LIN {X 0,Y 470.205,Z 358.727,A -85,B 0,C 180,E1 -7723.342,E2 -7723.342} C_VEL
LIN {X 0,Y 469.487,Z 370.693,A -85,B 0,C 180,E1 -7724.591,E2 -7724.591} C_VEL
LIN {X 0,Y 468.899,Z 381.216,A -85,B 0,C 180,E1 -7725.904,E2 -7725.904} C_VEL
LIN {X 0,Y 468.341,Z 390.427,A -85,B 0,C 180,E1 -7727.265,E2 -7727.265} C_VEL
LIN {X 0,Y 467.874,Z 398.79,A -85,B 0,C 180,E1 -7728.739,E2 -7728.739} C_VEL
LIN {X 0,Y 467.533,Z 405.048,A -85,B 0,C 180,E1 -7730.046,E2 -7730.046} C_VEL
LIN {X 0,Y 467.216,Z 411.873,A -85,B 0,C 180,E1 -7731.784,E2 -7731.784} C_VEL
LIN {X 0,Y 467.007,Z 416.636,A -85,B 0,C 180,E1 -7733.332,E2 -7733.332} C_VEL
LIN {X 0,Y 466.794,Z 420.207,A -85,B 0,C 180,E1 -7734.817,E2 -7734.817} C_VEL
LIN {X 0,Y 466.834,Z 423.167,A -85,B 0,C 180,E1 -7736.548,E2 -7736.548} C_VEL
LIN {X 0,Y 466.699,Z 424.922,A -85,B 0,C 180,E1 -7738.274,E2 -7738.274} C_VEL
LIN {X 0,Y 466.612,Z 425.477,A -85,B 0,C 180,E1 -7740,E2 -7740} C_VEL
LIN {X 0,Y 466.699,Z 424.809,A -85,B 0,C 180,E1 -7741.726,E2 -7741.726} C_VEL
LIN {X 0,Y 466.823,Z 422.958,A -85,B 0,C 180,E1 -7743.453,E2 -7743.453} C_VEL
LIN {X 0,Y 466.783,Z 419.896,A -85,B 0,C 180,E1 -7745.183,E2 -7745.183} C_VEL
LIN {X 0,Y 466.969,Z 416.065,A -85,B 0,C 180,E1 -7746.733,E2 -7746.733} C_VEL
LIN {X 0,Y 467.137,Z 411.402,A -85,B 0,C 180,E1 -7748.217,E2 -7748.217} C_VEL
LIN {X 0,Y 467.418,Z 404.499,A -85,B 0,C 180,E1 -7749.957,E2 -7749.957} C_VEL
LIN {X 0,Y 467.832,Z 397.038,A -85,B 0,C 180,E1 -7751.482,E2 -7751.482} C_VEL
LIN {X 0,Y 468.246,Z 388.039,A -85,B 0,C 180,E1 -7753.011,E2 -7753.011} C_VEL
LIN {X 0,Y 468.878,Z 377.174,A -85,B 0,C 180,E1 -7754.541,E2 -7754.541} C_VEL
LIN {X 0,Y 469.527,Z 365.967,A -85,B 0,C 180,E1 -7755.853,E2 -7755.853} C_VEL
LIN {X 0,Y 470.209,Z 354.013,A -85,B 0,C 180,E1 -7757.027,E2 -7757.027} C_VEL
LIN {X 0,Y 470.969,Z 340.123,A -85,B 0,C 180,E1 -7758.15,E2 -7758.15} C_VEL
LIN {X 0,Y 471.618,Z 326.912,A -85,B 0,C 180,E1 -7759.025,E2 -7759.025} C_VEL
LIN {X 0,Y 472.295,Z 312.467,A -85,B 0,C 180,E1 -7759.788,E2 -7759.788} C_VEL
LIN {X 0,Y 472.767,Z 297.672,A -85,B 0,C 180,E1 -7760.391,E2 -7760.391} C_VEL
LIN {X 0,Y 473.123,Z 282.745,A -85,B 0,C 180,E1 -7760.829,E2 -7760.829} C_VEL
LIN {X 0,Y 473.547,Z 255.622,A -85,B 0,C 180,E1 -7761.322,E2 -7761.322} C_VEL
LIN {X 0,Y 475.612,Z 134.89,A -85,B 0,C 180,E1 -7763.422,E2 -7763.422} C_VEL
LIN {X 0,Y 468.054,Z 114.952,A -85,B 0,C 180,E1 -7764.181,E2 -7764.181} C_VEL
LIN {X 0,Y 467.613,Z 112.864,A -85,B 0,C 180,E1 -7764.532,E2 -7764.532} C_VEL
LIN {X 0,Y 467.563,Z 112.87,A -85,B 0,C 180,E1 -7767.773,E2 -7767.773} C_VEL
LIN {X 0,Y 467.567,Z 112.867,A -85,B 0,C 180,E1 -7771.044,E2 -7771.044} C_VEL
LIN {X 0,Y 467.578,Z 112.864,A -85,B 0,C 180,E1 -7774.24,E2 -7774.24} C_VEL
LIN {X 0,Y 467.544,Z 112.871,A -85,B 0,C 180,E1 -7777.186,E2 -7777.186} C_VEL
LIN {X 0,Y 467.559,Z 112.865,A -85,B 0,C 180,E1 -7780.267,E2 -7780.267} C_VEL
LIN {X 0,Y 467.548,Z 112.866,A -85,B 0,C 180,E1 -7783.746,E2 -7783.746} C_VEL
LIN {X 0,Y 467.546,Z 112.852,A -85,B 0,C 180,E1 -7786.254,E2 -7786.254} C_VEL
LIN {X 0,Y 467.559,Z 112.867,A -85,B 0,C 180,E1 -7789.733,E2 -7789.733} C_VEL
LIN {X 0,Y 467.545,Z 112.869,A -85,B 0,C 180,E1 -7792.815,E2 -7792.815} C_VEL
LIN {X 0,Y 467.549,Z 112.855,A -85,B 0,C 180,E1 -7794.076,E2 -7794.076} C_VEL
LIN {X 0,Y 466.939,Z 112.935,A -85,B 0,C 180,E1 -7794.794,E2 -7794.794} C_VEL
LIN {X 0,Y 464.105,Z 113.293,A -85,B 0,C 180,E1 -7795.962,E2 -7795.962} C_VEL
LIN {X 0,Y 461.665,Z 113.603,A -85,B 0,C 180,E1 -7796.903,E2 -7796.903} C_VEL
LIN {X 0,Y 460.603,Z 113.733,A -85,B 0,C 180,E1 -7797.631,E2 -7797.631} C_VEL
LIN {X 0,Y 460.51,Z 113.743,A -85,B 0,C 180,E1 -7797.877,E2 -7797.877} C_VEL
LIN {X 0,Y 460.518,Z 113.738,A -85,B 0,C 180,E1 -7800.767,E2 -7800.767} C_VEL
LIN {X 0,Y 460.521,Z 113.743,A -85,B 0,C 180,E1 -7803.732,E2 -7803.732} C_VEL
LIN {X 0,Y 460.544,Z 113.737,A -85,B 0,C 180,E1 -7806.624,E2 -7806.624} C_VEL
LIN {X 0,Y 460.542,Z 113.737,A -85,B 0,C 180,E1 -7809.452,E2 -7809.452} C_VEL
LIN {X 0,Y 460.527,Z 113.745,A -85,B 0,C 180,E1 -7812.229,E2 -7812.229} C_VEL
LIN {X 0,Y 460.548,Z 113.743,A -85,B 0,C 180,E1 -7814.964,E2 -7814.964} C_VEL
LIN {X 0,Y 460.612,Z 113.736,A -85,B 0,C 180,E1 -7818.559,E2 -7818.559} C_VEL
LIN {X 0,Y 460.626,Z 113.732,A -85,B 0,C 180,E1 -7822.107,E2 -7822.107} C_VEL
LIN {X 0,Y 460.672,Z 113.729,A -85,B 0,C 180,E1 -7824.748,E2 -7824.748} C_VEL
LIN {X 0,Y 460.758,Z 113.718,A -85,B 0,C 180,E1 -7827.377,E2 -7827.377} C_VEL
LIN {X 0,Y 460.715,Z 113.854,A -85,B 0,C 180,E1 -7828.306,E2 -7828.306} C_VEL
LIN {X 0,Y 463.866,Z 127.486,A -85,B 0,C 180,E1 -7830.46,E2 -7830.46} C_VEL
LIN {X 0,Y 464.926,Z 132.74,A -85,B 0,C 180,E1 -7831.28,E2 -7831.28} C_VEL
LIN {X 0,Y 464.725,Z 142.504,A -85,B 0,C 180,E1 -7832.646,E2 -7832.646} C_VEL
LIN {X 0,Y 469.356,Z 164.409,A -85,B 0,C 180,E1 -7833.26,E2 -7833.26} C_VEL
LIN {X 0,Y 467.464,Z 308.671,A -85,B 0,C 180,E1 -7835.554,E2 -7835.554} C_VEL
LIN {X 0,Y 467.063,Z 323.846,A -85,B 0,C 180,E1 -7835.965,E2 -7835.965} C_VEL
LIN {X 0,Y 466.453,Z 338.982,A -85,B 0,C 180,E1 -7836.556,E2 -7836.556} C_VEL
LIN {X 0,Y 465.768,Z 352.68,A -85,B 0,C 180,E1 -7837.26,E2 -7837.26} C_VEL
LIN {X 0,Y 464.914,Z 366.405,A -85,B 0,C 180,E1 -7838.147,E2 -7838.147} C_VEL
LIN {X 0,Y 464.107,Z 378.997,A -85,B 0,C 180,E1 -7839.149,E2 -7839.149} C_VEL
LIN {X 0,Y 463.263,Z 390.836,A -85,B 0,C 180,E1 -7840.28,E2 -7840.28} C_VEL
LIN {X 0,Y 462.424,Z 402.5,A -85,B 0,C 180,E1 -7841.617,E2 -7841.617} C_VEL
LIN {X 0,Y 461.673,Z 412.766,A -85,B 0,C 180,E1 -7843.025,E2 -7843.025} C_VEL
LIN {X 0,Y 461.03,Z 422.16,A -85,B 0,C 180,E1 -7844.568,E2 -7844.568} C_VEL
LIN {X 0,Y 460.56,Z 429.373,A -85,B 0,C 180,E1 -7845.978,E2 -7845.978} C_VEL
LIN {X 0,Y 460.148,Z 436.979,A -85,B 0,C 180,E1 -7847.786,E2 -7847.786} C_VEL
LIN {X 0,Y 459.856,Z 443.115,A -85,B 0,C 180,E1 -7849.647,E2 -7849.647} C_VEL
LIN {X 0,Y 459.632,Z 447.79,A -85,B 0,C 180,E1 -7851.529,E2 -7851.529} C_VEL
LIN {X 0,Y 459.464,Z 451.071,A -85,B 0,C 180,E1 -7853.434,E2 -7853.434} C_VEL
LIN {X 0,Y 459.416,Z 452.973,A -85,B 0,C 180,E1 -7855.362,E2 -7855.362} C_VEL
LIN {X 0,Y 459.426,Z 453.492,A -85,B 0,C 180,E1 -7857.317,E2 -7857.317} C_VEL
LIN {X 0,Y 459.45,Z 452.559,A -85,B 0,C 180,E1 -7859.319,E2 -7859.319} C_VEL
LIN {X 0,Y 459.534,Z 450.116,A -85,B 0,C 180,E1 -7861.331,E2 -7861.331} C_VEL
LIN {X 0,Y 459.649,Z 447.476,A -85,B 0,C 180,E1 -7862.759,E2 -7862.759} C_VEL
LIN {X 0,Y 459.815,Z 443.254,A -85,B 0,C 180,E1 -7864.439,E2 -7864.439} C_VEL
LIN {X 0,Y 460.136,Z 437.453,A -85,B 0,C 180,E1 -7866.215,E2 -7866.215} C_VEL
LIN {X 0,Y 460.508,Z 430.544,A -85,B 0,C 180,E1 -7867.899,E2 -7867.899} C_VEL
LIN {X 0,Y 461.041,Z 422.167,A -85,B 0,C 180,E1 -7869.567,E2 -7869.567} C_VEL
LIN {X 0,Y 461.744,Z 412.393,A -85,B 0,C 180,E1 -7871.17,E2 -7871.17} C_VEL
LIN {X 0,Y 462.565,Z 401.147,A -85,B 0,C 180,E1 -7872.689,E2 -7872.689} C_VEL
LIN {X 0,Y 463.356,Z 389.986,A -85,B 0,C 180,E1 -7873.948,E2 -7873.948} C_VEL
LIN {X 0,Y 464.296,Z 377.438,A -85,B 0,C 180,E1 -7875.123,E2 -7875.123} C_VEL
LIN {X 0,Y 465.113,Z 364.512,A -85,B 0,C 180,E1 -7876.125,E2 -7876.125} C_VEL
LIN {X 0,Y 465.98,Z 350.355,A -85,B 0,C 180,E1 -7877.009,E2 -7877.009} C_VEL
LIN {X 0,Y 466.709,Z 336.007,A -85,B 0,C 180,E1 -7877.711,E2 -7877.711} C_VEL
LIN {X 0,Y 467.223,Z 320.852,A -85,B 0,C 180,E1 -7878.265,E2 -7878.265} C_VEL
LIN {X 0,Y 467.643,Z 306.467,A -85,B 0,C 180,E1 -7878.621,E2 -7878.621} C_VEL
LIN {X 0,Y 469.619,Z 160.081,A -85,B 0,C 180,E1 -7880.948,E2 -7880.948} C_VEL
LIN {X 0,Y 466.099,Z 140.754,A -85,B 0,C 180,E1 -7881.491,E2 -7881.491} C_VEL
LIN {X 0,Y 466.266,Z 135.208,A -85,B 0,C 180,E1 -7882.104,E2 -7882.104} C_VEL
LIN {X 0,Y 462.6,Z 121.002,A -85,B 0,C 180,E1 -7883.914,E2 -7883.914} C_VEL
LIN {X 0,Y 460.536,Z 113.744,A -85,B 0,C 180,E1 -7884.871,E2 -7884.871} C_VEL
LIN {X 0,Y 460.534,Z 113.747,A -85,B 0,C 180,E1 -7887.715,E2 -7887.715} C_VEL
LIN {X 0,Y 460.542,Z 113.739,A -85,B 0,C 180,E1 -7890.769,E2 -7890.769} C_VEL
LIN {X 0,Y 460.566,Z 113.742,A -85,B 0,C 180,E1 -7893.735,E2 -7893.735} C_VEL
LIN {X 0,Y 460.57,Z 113.75,A -85,B 0,C 180,E1 -7895.369,E2 -7895.369} C_VEL
LIN {X 0,Y 460.779,Z 114.732,A -85,B 0,C 180,E1 -7895.514,E2 -7895.514} C_VEL
LIN {X 0,Y 469.062,Z 135.535,A -85,B 0,C 180,E1 -7896.336,E2 -7896.336} C_VEL
LIN {X 0,Y 466.423,Z 282.486,A -85,B 0,C 180,E1 -7898.977,E2 -7898.977} C_VEL
LIN {X 0,Y 466.028,Z 297.981,A -85,B 0,C 180,E1 -7899.434,E2 -7899.434} C_VEL
LIN {X 0,Y 465.501,Z 312.425,A -85,B 0,C 180,E1 -7900.026,E2 -7900.026} C_VEL
LIN {X 0,Y 464.802,Z 326.942,A -85,B 0,C 180,E1 -7900.8,E2 -7900.8} C_VEL
LIN {X 0,Y 464.134,Z 340.27,A -85,B 0,C 180,E1 -7901.687,E2 -7901.687} C_VEL
LIN {X 0,Y 463.457,Z 352.85,A -85,B 0,C 180,E1 -7902.706,E2 -7902.706} C_VEL
LIN {X 0,Y 462.676,Z 365.193,A -85,B 0,C 180,E1 -7903.906,E2 -7903.906} C_VEL
LIN {X 0,Y 462.018,Z 376.615,A -85,B 0,C 180,E1 -7905.238,E2 -7905.238} C_VEL
LIN {X 0,Y 461.33,Z 387.666,A -85,B 0,C 180,E1 -7906.79,E2 -7906.79} C_VEL
LIN {X 0,Y 460.873,Z 396.82,A -85,B 0,C 180,E1 -7908.343,E2 -7908.343} C_VEL
LIN {X 0,Y 460.423,Z 404.413,A -85,B 0,C 180,E1 -7909.89,E2 -7909.89} C_VEL
LIN {X 0,Y 460.104,Z 411.459,A -85,B 0,C 180,E1 -7911.656,E2 -7911.656} C_VEL
LIN {X 0,Y 459.861,Z 416.937,A -85,B 0,C 180,E1 -7913.408,E2 -7913.408} C_VEL
LIN {X 0,Y 459.736,Z 420.149,A -85,B 0,C 180,E1 -7914.737,E2 -7914.737} C_VEL
LIN {X 0,Y 459.76,Z 423.312,A -85,B 0,C 180,E1 -7916.494,E2 -7916.494} C_VEL
LIN {X 0,Y 459.638,Z 425.267,A -85,B 0,C 180,E1 -7918.247,E2 -7918.247} C_VEL
LIN {X 0,Y 459.545,Z 426.009,A -85,B 0,C 180,E1 -7920,E2 -7920} C_VEL
LIN {X 0,Y 459.639,Z 425.528,A -85,B 0,C 180,E1 -7921.752,E2 -7921.752} C_VEL
LIN {X 0,Y 459.777,Z 423.863,A -85,B 0,C 180,E1 -7923.505,E2 -7923.505} C_VEL
LIN {X 0,Y 459.749,Z 420.99,A -85,B 0,C 180,E1 -7925.262,E2 -7925.262} C_VEL
LIN {X 0,Y 460.008,Z 417.57,A -85,B 0,C 180,E1 -7926.749,E2 -7926.749} C_VEL
LIN {X 0,Y 460.19,Z 412.788,A -85,B 0,C 180,E1 -7928.342,E2 -7928.342} C_VEL
LIN {X 0,Y 460.528,Z 406.086,A -85,B 0,C 180,E1 -7930.107,E2 -7930.107} C_VEL
LIN {X 0,Y 460.97,Z 398.787,A -85,B 0,C 180,E1 -7931.654,E2 -7931.654} C_VEL
LIN {X 0,Y 461.482,Z 389.975,A -85,B 0,C 180,E1 -7933.205,E2 -7933.205} C_VEL
LIN {X 0,Y 462.121,Z 380.966,A -85,B 0,C 180,E1 -7934.533,E2 -7934.533} C_VEL
LIN {X 0,Y 462.797,Z 370.287,A -85,B 0,C 180,E1 -7935.863,E2 -7935.863} C_VEL
LIN {X 0,Y 463.608,Z 357.669,A -85,B 0,C 180,E1 -7937.173,E2 -7937.173} C_VEL
LIN {X 0,Y 464.377,Z 344.479,A -85,B 0,C 180,E1 -7938.302,E2 -7938.302} C_VEL
LIN {X 0,Y 465.093,Z 331.89,A -85,B 0,C 180,E1 -7939.187,E2 -7939.187} C_VEL
LIN {X 0,Y 465.707,Z 318.4,A -85,B 0,C 180,E1 -7939.964,E2 -7939.964} C_VEL
LIN {X 0,Y 466.334,Z 302.907,A -85,B 0,C 180,E1 -7940.654,E2 -7940.654} C_VEL
LIN {X 0,Y 466.798,Z 287.065,A -85,B 0,C 180,E1 -7941.165,E2 -7941.165} C_VEL
LIN {X 0,Y 467.313,Z 262.068,A -85,B 0,C 180,E1 -7941.678,E2 -7941.678} C_VEL
LIN {X 0,Y 469.548,Z 178.96,A -85,B 0,C 180,E1 -7943.33,E2 -7943.33} C_VEL
LIN {X 0,Y 470.871,Z 139.064,A -85,B 0,C 180,E1 -7944.172,E2 -7944.172} C_VEL
LIN {X 0,Y 465.458,Z 127.422,A -85,B 0,C 180,E1 -7944.861,E2 -7944.861} C_VEL
LIN {X 0,Y 462.823,Z 122.223,A -85,B 0,C 180,E1 -7945.225,E2 -7945.225} C_VEL
LIN {X 0,Y 460.525,Z 113.749,A -85,B 0,C 180,E1 -7947.45,E2 -7947.45} C_VEL
LIN {X 0,Y 460.504,Z 113.75,A -85,B 0,C 180,E1 -7950.24,E2 -7950.24} C_VEL
LIN {X 0,Y 460.516,Z 113.748,A -85,B 0,C 180,E1 -7953.326,E2 -7953.326} C_VEL
LIN {X 0,Y 460.472,Z 113.752,A -85,B 0,C 180,E1 -7956.53,E2 -7956.53} C_VEL
LIN {X 0,Y 460.513,Z 113.748,A -85,B 0,C 180,E1 -7959.864,E2 -7959.864} C_VEL
LIN {X 0,Y 460.461,Z 113.754,A -85,B 0,C 180,E1 -7962.893,E2 -7962.893} C_VEL
LIN {X 0,Y 460.502,Z 113.748,A -85,B 0,C 180,E1 -7965.831,E2 -7965.831} C_VEL
LIN {X 0,Y 460.513,Z 113.749,A -85,B 0,C 180,E1 -7968.987,E2 -7968.987} C_VEL
LIN {X 0,Y 460.497,Z 113.751,A -85,B 0,C 180,E1 -7972.376,E2 -7972.376} C_VEL
LIN {X 0,Y 460.534,Z 113.747,A -85,B 0,C 180,E1 -7975.623,E2 -7975.623} C_VEL
LIN {X 0,Y 460.531,Z 113.873,A -85,B 0,C 180,E1 -7976.854,E2 -7976.854} C_VEL
LIN {X 0,Y 463.777,Z 124.861,A -85,B 0,C 180,E1 -7979.198,E2 -7979.198} C_VEL
LIN {X 0,Y 466.239,Z 135.335,A -85,B 0,C 180,E1 -7981.16,E2 -7981.16} C_VEL
LIN {X 0,Y 466.332,Z 138.39,A -85,B 0,C 180,E1 -7981.658,E2 -7981.658} C_VEL
LIN {X 0,Y 464.916,Z 155.637,A -85,B 0,C 180,E1 -7984.24,E2 -7984.24} C_VEL
LIN {X 0,Y 464.589,Z 160.323,A -85,B 0,C 180,E1 -7984.925,E2 -7984.925} C_VEL
LIN {X 0,Y 468.206,Z 179.445,A -85,B 0,C 180,E1 -7985.649,E2 -7985.649} C_VEL
LIN {X 0,Y 469.863,Z 191.952,A -85,B 0,C 180,E1 -7986.049,E2 -7986.049} C_VEL
LIN {X 0,Y 467.42,Z 282.385,A -85,B 0,C 180,E1 -7987.862,E2 -7987.862} C_VEL
LIN {X 0,Y 466.4,Z 330.968,A -85,B 0,C 180,E1 -7988.799,E2 -7988.799} C_VEL
LIN {X 0,Y 465.612,Z 350.742,A -85,B 0,C 180,E1 -7989.39,E2 -7989.39} C_VEL
LIN {X 0,Y 465.03,Z 366.077,A -85,B 0,C 180,E1 -7990.005,E2 -7990.005} C_VEL
LIN {X 0,Y 464.275,Z 380.562,A -85,B 0,C 180,E1 -7990.777,E2 -7990.777} C_VEL
LIN {X 0,Y 463.575,Z 393.745,A -85,B 0,C 180,E1 -7991.665,E2 -7991.665} C_VEL
LIN {X 0,Y 462.845,Z 405.936,A -85,B 0,C 180,E1 -7992.663,E2 -7992.663} C_VEL
LIN {X 0,Y 461.989,Z 418.546,A -85,B 0,C 180,E1 -7993.912,E2 -7993.912} C_VEL
LIN {X 0,Y 461.396,Z 429.488,A -85,B 0,C 180,E1 -7995.218,E2 -7995.218} C_VEL
LIN {X 0,Y 460.854,Z 438.906,A -85,B 0,C 180,E1 -7996.552,E2 -7996.552} C_VEL
LIN {X 0,Y 460.304,Z 448.353,A -85,B 0,C 180,E1 -7998.146,E2 -7998.146} C_VEL
LIN {X 0,Y 460.037,Z 455.754,A -85,B 0,C 180,E1 -7999.659,E2 -7999.659} C_VEL
LIN {X 0,Y 459.802,Z 462.035,A -85,B 0,C 180,E1 -8001.208,E2 -8001.208} C_VEL
LIN {X 0,Y 459.725,Z 467.769,A -85,B 0,C 180,E1 -8002.975,E2 -8002.975} C_VEL
LIN {X 0,Y 459.626,Z 472.092,A -85,B 0,C 180,E1 -8004.736,E2 -8004.736} C_VEL
LIN {X 0,Y 459.595,Z 475.12,A -85,B 0,C 180,E1 -8006.493,E2 -8006.493} C_VEL
LIN {X 0,Y 459.598,Z 476.93,A -85,B 0,C 180,E1 -8008.247,E2 -8008.247} C_VEL
LIN {X 0,Y 459.536,Z 477.546,A -85,B 0,C 180,E1 -8010,E2 -8010} C_VEL
LIN {X 0,Y 459.597,Z 476.948,A -85,B 0,C 180,E1 -8011.753,E2 -8011.753} C_VEL
LIN {X 0,Y 459.608,Z 475.152,A -85,B 0,C 180,E1 -8013.507,E2 -8013.507} C_VEL
LIN {X 0,Y 459.63,Z 472.125,A -85,B 0,C 180,E1 -8015.264,E2 -8015.264} C_VEL
LIN {X 0,Y 459.727,Z 467.802,A -85,B 0,C 180,E1 -8017.025,E2 -8017.025} C_VEL
LIN {X 0,Y 459.802,Z 462.075,A -85,B 0,C 180,E1 -8018.792,E2 -8018.792} C_VEL
LIN {X 0,Y 460.128,Z 454.78,A -85,B 0,C 180,E1 -8020.561,E2 -8020.561} C_VEL
LIN {X 0,Y 460.382,Z 446.748,A -85,B 0,C 180,E1 -8022.146,E2 -8022.146} C_VEL
LIN {X 0,Y 460.882,Z 437.413,A -85,B 0,C 180,E1 -8023.672,E2 -8023.672} C_VEL
LIN {X 0,Y 461.45,Z 427.686,A -85,B 0,C 180,E1 -8025.006,E2 -8025.006} C_VEL
LIN {X 0,Y 462.107,Z 416.662,A -85,B 0,C 180,E1 -8026.278,E2 -8026.278} C_VEL
LIN {X 0,Y 462.801,Z 404.49,A -85,B 0,C 180,E1 -8027.453,E2 -8027.453} C_VEL
LIN {X 0,Y 463.626,Z 391.995,A -85,B 0,C 180,E1 -8028.448,E2 -8028.448} C_VEL
LIN {X 0,Y 464.369,Z 378.323,A -85,B 0,C 180,E1 -8029.334,E2 -8029.334} C_VEL
LIN {X 0,Y 465.059,Z 364.285,A -85,B 0,C 180,E1 -8030.051,E2 -8030.051} C_VEL
LIN {X 0,Y 465.774,Z 346.56,A -85,B 0,C 180,E1 -8030.748,E2 -8030.748} C_VEL
LIN {X 0,Y 466.243,Z 330.73,A -85,B 0,C 180,E1 -8031.184,E2 -8031.184} C_VEL
LIN {X 0,Y 468.656,Z 202.97,A -85,B 0,C 180,E1 -8033.474,E2 -8033.474} C_VEL
LIN {X 0,Y 468.982,Z 186.436,A -85,B 0,C 180,E1 -8033.833,E2 -8033.833} C_VEL
LIN {X 0,Y 465.653,Z 160.353,A -85,B 0,C 180,E1 -8034.701,E2 -8034.701} C_VEL
LIN {X 0,Y 466.909,Z 137.343,A -85,B 0,C 180,E1 -8037.197,E2 -8037.197} C_VEL
LIN {X 0,Y 462.077,Z 119.489,A -85,B 0,C 180,E1 -8039.494,E2 -8039.494} C_VEL
LIN {X 0,Y 460.535,Z 113.746,A -85,B 0,C 180,E1 -8040.27,E2 -8040.27} C_VEL
LIN {X 0,Y 460.515,Z 113.748,A -85,B 0,C 180,E1 -8043.326,E2 -8043.326} C_VEL
LIN {X 0,Y 460.471,Z 113.754,A -85,B 0,C 180,E1 -8046.53,E2 -8046.53} C_VEL
LIN {X 0,Y 460.512,Z 113.746,A -85,B 0,C 180,E1 -8049.865,E2 -8049.865} C_VEL
LIN {X 0,Y 460.461,Z 113.755,A -85,B 0,C 180,E1 -8052.894,E2 -8052.894} C_VEL
LIN {X 0,Y 460.502,Z 113.743,A -85,B 0,C 180,E1 -8055.832,E2 -8055.832} C_VEL
LIN {X 0,Y 460.514,Z 113.745,A -85,B 0,C 180,E1 -8058.987,E2 -8058.987} C_VEL
LIN {X 0,Y 460.497,Z 113.75,A -85,B 0,C 180,E1 -8062.377,E2 -8062.377} C_VEL
LIN {X 0,Y 460.535,Z 113.743,A -85,B 0,C 180,E1 -8065.623,E2 -8065.623} C_VEL
LIN {X 0,Y 460.537,Z 113.746,A -85,B 0,C 180,E1 -8068.745,E2 -8068.745} C_VEL
LIN {X 0,Y 460.531,Z 113.748,A -85,B 0,C 180,E1 -8072.266,E2 -8072.266} C_VEL
LIN {X 0,Y 460.539,Z 113.891,A -85,B 0,C 180,E1 -8073.84,E2 -8073.84} C_VEL
LIN {X 0,Y 462.385,Z 119.757,A -85,B 0,C 180,E1 -8074.851,E2 -8074.851} C_VEL
LIN {X 0,Y 468.701,Z 132.928,A -85,B 0,C 180,E1 -8075.669,E2 -8075.669} C_VEL
LIN {X 0,Y 470.74,Z 137.876,A -85,B 0,C 180,E1 -8075.936,E2 -8075.936} C_VEL
LIN {X 0,Y 468.083,Z 226.35,A -85,B 0,C 180,E1 -8077.75,E2 -8077.75} C_VEL
LIN {X 0,Y 466.781,Z 285.261,A -85,B 0,C 180,E1 -8078.901,E2 -8078.901} C_VEL
LIN {X 0,Y 466.28,Z 301.493,A -85,B 0,C 180,E1 -8079.4,E2 -8079.4} C_VEL
LIN {X 0,Y 465.757,Z 316.216,A -85,B 0,C 180,E1 -8080.038,E2 -8080.038} C_VEL
LIN {X 0,Y 465.121,Z 330.113,A -85,B 0,C 180,E1 -8080.814,E2 -8080.814} C_VEL
LIN {X 0,Y 464.351,Z 344.421,A -85,B 0,C 180,E1 -8081.811,E2 -8081.811} C_VEL
LIN {X 0,Y 463.594,Z 356.511,A -85,B 0,C 180,E1 -8082.832,E2 -8082.832} C_VEL
LIN {X 0,Y 462.747,Z 369.234,A -85,B 0,C 180,E1 -8084.135,E2 -8084.135} C_VEL
LIN {X 0,Y 462.156,Z 380.059,A -85,B 0,C 180,E1 -8085.469,E2 -8085.469} C_VEL
LIN {X 0,Y 461.53,Z 389.205,A -85,B 0,C 180,E1 -8086.797,E2 -8086.797} C_VEL
LIN {X 0,Y 460.987,Z 398.127,A -85,B 0,C 180,E1 -8088.346,E2 -8088.346} C_VEL
LIN {X 0,Y 460.539,Z 405.491,A -85,B 0,C 180,E1 -8089.893,E2 -8089.893} C_VEL
LIN {X 0,Y 460.18,Z 412.311,A -85,B 0,C 180,E1 -8091.658,E2 -8091.658} C_VEL
LIN {X 0,Y 459.964,Z 417.265,A -85,B 0,C 180,E1 -8093.298,E2 -8093.298} C_VEL
LIN {X 0,Y 459.738,Z 420.64,A -85,B 0,C 180,E1 -8094.738,E2 -8094.738} C_VEL
LIN {X 0,Y 459.765,Z 423.589,A -85,B 0,C 180,E1 -8096.495,E2 -8096.495} C_VEL
LIN {X 0,Y 459.639,Z 425.328,A -85,B 0,C 180,E1 -8098.248,E2 -8098.248} C_VEL
LIN {X 0,Y 459.543,Z 425.869,A -85,B 0,C 180,E1 -8100,E2 -8100} C_VEL
LIN {X 0,Y 459.637,Z 425.178,A -85,B 0,C 180,E1 -8101.753,E2 -8101.753} C_VEL
LIN {X 0,Y 459.752,Z 423.296,A -85,B 0,C 180,E1 -8103.506,E2 -8103.506} C_VEL
LIN {X 0,Y 459.729,Z 420.196,A -85,B 0,C 180,E1 -8105.263,E2 -8105.263} C_VEL
LIN {X 0,Y 459.921,Z 415.793,A -85,B 0,C 180,E1 -8107.022,E2 -8107.022} C_VEL
LIN {X 0,Y 460.143,Z 409.989,A -85,B 0,C 180,E1 -8108.786,E2 -8108.786} C_VEL
LIN {X 0,Y 460.465,Z 402.615,A -85,B 0,C 180,E1 -8110.554,E2 -8110.554} C_VEL
LIN {X 0,Y 460.921,Z 394.673,A -85,B 0,C 180,E1 -8112.103,E2 -8112.103} C_VEL
LIN {X 0,Y 461.438,Z 385.101,A -85,B 0,C 180,E1 -8113.655,E2 -8113.655} C_VEL
LIN {X 0,Y 462.059,Z 375.307,A -85,B 0,C 180,E1 -8114.986,E2 -8114.986} C_VEL
LIN {X 0,Y 462.777,Z 363.644,A -85,B 0,C 180,E1 -8116.317,E2 -8116.317} C_VEL
LIN {X 0,Y 463.519,Z 350.687,A -85,B 0,C 180,E1 -8117.548,E2 -8117.548} C_VEL
LIN {X 0,Y 464.205,Z 338.078,A -85,B 0,C 180,E1 -8118.539,E2 -8118.539} C_VEL
LIN {X 0,Y 464.921,Z 324.287,A -85,B 0,C 180,E1 -8119.425,E2 -8119.425} C_VEL
LIN {X 0,Y 465.578,Z 309.007,A -85,B 0,C 180,E1 -8120.201,E2 -8120.201} C_VEL
LIN {X 0,Y 466.048,Z 293.672,A -85,B 0,C 180,E1 -8120.787,E2 -8120.787} C_VEL
LIN {X 0,Y 466.444,Z 277.954,A -85,B 0,C 180,E1 -8121.2,E2 -8121.2} C_VEL
LIN {X 0,Y 469.059,Z 137.414,A -85,B 0,C 180,E1 -8123.698,E2 -8123.698} C_VEL
LIN {X 0,Y 468.467,Z 134.85,A -85,B 0,C 180,E1 -8123.776,E2 -8123.776} C_VEL
LIN {X 0,Y 460.88,Z 115.188,A -85,B 0,C 180,E1 -8124.551,E2 -8124.551} C_VEL
LIN {X 0,Y 460.553,Z 113.743,A -85,B 0,C 180,E1 -8124.813,E2 -8124.813} C_VEL
LIN {X 0,Y 460.516,Z 113.746,A -85,B 0,C 180,E1 -8128.236,E2 -8128.236} C_VEL
LIN {X 0,Y 460.522,Z 113.746,A -85,B 0,C 180,E1 -8131.283,E2 -8131.283} C_VEL
LIN {X 0,Y 460.523,Z 113.742,A -85,B 0,C 180,E1 -8134.504,E2 -8134.504} C_VEL
LIN {X 0,Y 460.5,Z 113.75,A -85,B 0,C 180,E1 -8137.624,E2 -8137.624} C_VEL
LIN {X 0,Y 460.517,Z 113.745,A -85,B 0,C 180,E1 -8141.013,E2 -8141.013} C_VEL
LIN {X 0,Y 460.514,Z 113.74,A -85,B 0,C 180,E1 -8144.59,E2 -8144.59} C_VEL
LIN {X 0,Y 460.477,Z 113.743,A -85,B 0,C 180,E1 -8147.813,E2 -8147.813} C_VEL
LIN {X 0,Y 460.515,Z 113.743,A -85,B 0,C 180,E1 -8150.136,E2 -8150.136} C_VEL
LIN {X 0,Y 460.475,Z 113.739,A -85,B 0,C 180,E1 -8153.47,E2 -8153.47} C_VEL
LIN {X 0,Y 460.519,Z 113.743,A -85,B 0,C 180,E1 -8156.674,E2 -8156.674} C_VEL
LIN {X 0,Y 460.51,Z 113.743,A -85,B 0,C 180,E1 -8157.877,E2 -8157.877} C_VEL
LIN {X 0,Y 459.825,Z 113.832,A -85,B 0,C 180,E1 -8158.608,E2 -8158.608} C_VEL
LIN {X 0,Y 456.959,Z 114.185,A -85,B 0,C 180,E1 -8159.793,E2 -8159.793} C_VEL
LIN {X 0,Y 454.555,Z 114.483,A -85,B 0,C 180,E1 -8160.75,E2 -8160.75} C_VEL
LIN {X 0,Y 453.538,Z 114.611,A -85,B 0,C 180,E1 -8161.489,E2 -8161.489} C_VEL
LIN {X 0,Y 453.462,Z 114.619,A -85,B 0,C 180,E1 -8161.739,E2 -8161.739} C_VEL
LIN {X 0,Y 453.496,Z 114.62,A -85,B 0,C 180,E1 -8164.283,E2 -8164.283} C_VEL
LIN {X 0,Y 453.476,Z 114.622,A -85,B 0,C 180,E1 -8167.204,E2 -8167.204} C_VEL
LIN {X 0,Y 453.498,Z 114.615,A -85,B 0,C 180,E1 -8170.066,E2 -8170.066} C_VEL
LIN {X 0,Y 453.475,Z 114.621,A -85,B 0,C 180,E1 -8172.875,E2 -8172.875} C_VEL
LIN {X 0,Y 453.498,Z 114.619,A -85,B 0,C 180,E1 -8175.643,E2 -8175.643} C_VEL
LIN {X 0,Y 453.561,Z 114.616,A -85,B 0,C 180,E1 -8178.379,E2 -8178.379} C_VEL
LIN {X 0,Y 453.564,Z 114.61,A -85,B 0,C 180,E1 -8181.086,E2 -8181.086} C_VEL
LIN {X 0,Y 453.631,Z 114.604,A -85,B 0,C 180,E1 -8183.774,E2 -8183.774} C_VEL
LIN {X 0,Y 453.689,Z 114.602,A -85,B 0,C 180,E1 -8187.781,E2 -8187.781} C_VEL
LIN {X 0,Y 453.729,Z 114.857,A -85,B 0,C 180,E1 -8188.003,E2 -8188.003} C_VEL
LIN {X 0,Y 456.825,Z 128.141,A -85,B 0,C 180,E1 -8190.133,E2 -8190.133} C_VEL
LIN {X 0,Y 458.173,Z 135.454,A -85,B 0,C 180,E1 -8191.273,E2 -8191.273} C_VEL
LIN {X 0,Y 457.986,Z 142.634,A -85,B 0,C 180,E1 -8192.275,E2 -8192.275} C_VEL
LIN {X 0,Y 462.797,Z 164.858,A -85,B 0,C 180,E1 -8192.918,E2 -8192.918} C_VEL
LIN {X 0,Y 460.877,Z 307.956,A -85,B 0,C 180,E1 -8195.222,E2 -8195.222} C_VEL
LIN {X 0,Y 460.434,Z 323.473,A -85,B 0,C 180,E1 -8195.639,E2 -8195.639} C_VEL
LIN {X 0,Y 459.818,Z 338.413,A -85,B 0,C 180,E1 -8196.222,E2 -8196.222} C_VEL
LIN {X 0,Y 459.049,Z 352.935,A -85,B 0,C 180,E1 -8196.975,E2 -8196.975} C_VEL
LIN {X 0,Y 458.223,Z 365.957,A -85,B 0,C 180,E1 -8197.823,E2 -8197.823} C_VEL
LIN {X 0,Y 457.307,Z 378.703,A -85,B 0,C 180,E1 -8198.84,E2 -8198.84} C_VEL
LIN {X 0,Y 456.431,Z 391.056,A -85,B 0,C 180,E1 -8200.037,E2 -8200.037} C_VEL
LIN {X 0,Y 455.558,Z 402.338,A -85,B 0,C 180,E1 -8201.344,E2 -8201.344} C_VEL
LIN {X 0,Y 454.76,Z 412.8,A -85,B 0,C 180,E1 -8202.794,E2 -8202.794} C_VEL
LIN {X 0,Y 454.073,Z 422.108,A -85,B 0,C 180,E1 -8204.338,E2 -8204.338} C_VEL
LIN {X 0,Y 453.48,Z 430.751,A -85,B 0,C 180,E1 -8206.08,E2 -8206.08} C_VEL
LIN {X 0,Y 453.122,Z 437,A -85,B 0,C 180,E1 -8207.605,E2 -8207.605} C_VEL
LIN {X 0,Y 452.787,Z 443.183,A -85,B 0,C 180,E1 -8209.494,E2 -8209.494} C_VEL
LIN {X 0,Y 452.586,Z 447.671,A -85,B 0,C 180,E1 -8211.296,E2 -8211.296} C_VEL
LIN {X 0,Y 452.355,Z 451.47,A -85,B 0,C 180,E1 -8213.557,E2 -8213.557} C_VEL
LIN {X 0,Y 452.297,Z 452.77,A -85,B 0,C 180,E1 -8214.805,E2 -8214.805} C_VEL
LIN {X 0,Y 452.292,Z 453.676,A -85,B 0,C 180,E1 -8216.784,E2 -8216.784} C_VEL
LIN {X 0,Y 452.318,Z 453.164,A -85,B 0,C 180,E1 -8218.795,E2 -8218.795} C_VEL
LIN {X 0,Y 452.381,Z 452.354,A -85,B 0,C 180,E1 -8219.811,E2 -8219.811} C_VEL
LIN {X 0,Y 452.456,Z 450.439,A -85,B 0,C 180,E1 -8221.315,E2 -8221.315} C_VEL
LIN {X 0,Y 452.574,Z 447.3,A -85,B 0,C 180,E1 -8223.011,E2 -8223.011} C_VEL
LIN {X 0,Y 452.782,Z 443.197,A -85,B 0,C 180,E1 -8224.648,E2 -8224.648} C_VEL
LIN {X 0,Y 453.061,Z 438.095,A -85,B 0,C 180,E1 -8226.231,E2 -8226.231} C_VEL
LIN {X 0,Y 453.491,Z 431.052,A -85,B 0,C 180,E1 -8227.997,E2 -8227.997} C_VEL
LIN {X 0,Y 454.028,Z 422.797,A -85,B 0,C 180,E1 -8229.681,E2 -8229.681} C_VEL
LIN {X 0,Y 454.714,Z 414.167,A -85,B 0,C 180,E1 -8231.141,E2 -8231.141} C_VEL
LIN {X 0,Y 455.51,Z 404.027,A -85,B 0,C 180,E1 -8232.584,E2 -8232.584} C_VEL
LIN {X 0,Y 456.309,Z 393.256,A -85,B 0,C 180,E1 -8233.875,E2 -8233.875} C_VEL
LIN {X 0,Y 457.322,Z 380.551,A -85,B 0,C 180,E1 -8235.14,E2 -8235.14} C_VEL
LIN {X 0,Y 458.196,Z 368.559,A -85,B 0,C 180,E1 -8236.129,E2 -8236.129} C_VEL
LIN {X 0,Y 459.09,Z 354.506,A -85,B 0,C 180,E1 -8237.079,E2 -8237.079} C_VEL
LIN {X 0,Y 459.877,Z 339.71,A -85,B 0,C 180,E1 -8237.867,E2 -8237.867} C_VEL
LIN {X 0,Y 460.535,Z 324.752,A -85,B 0,C 180,E1 -8238.464,E2 -8238.464} C_VEL
LIN {X 0,Y 460.986,Z 310.334,A -85,B 0,C 180,E1 -8238.866,E2 -8238.866} C_VEL
LIN {X 0,Y 461.501,Z 274.997,A -85,B 0,C 180,E1 -8239.464,E2 -8239.464} C_VEL
LIN {X 0,Y 463.152,Z 160.953,A -85,B 0,C 180,E1 -8241.297,E2 -8241.297} C_VEL
LIN {X 0,Y 459.475,Z 141.081,A -85,B 0,C 180,E1 -8241.861,E2 -8241.861} C_VEL
LIN {X 0,Y 459.608,Z 137.252,A -85,B 0,C 180,E1 -8242.291,E2 -8242.291} C_VEL
LIN {X 0,Y 455.424,Z 121.16,A -85,B 0,C 180,E1 -8244.37,E2 -8244.37} C_VEL
LIN {X 0,Y 453.515,Z 114.618,A -85,B 0,C 180,E1 -8245.262,E2 -8245.262} C_VEL
LIN {X 0,Y 453.468,Z 114.623,A -85,B 0,C 180,E1 -8248.475,E2 -8248.475} C_VEL
LIN {X 0,Y 453.535,Z 114.617,A -85,B 0,C 180,E1 -8252.04,E2 -8252.04} C_VEL
LIN {X 0,Y 453.568,Z 114.799,A -85,B 0,C 180,E1 -8255.116,E2 -8255.116} C_VEL
LIN {X 0,Y 462.415,Z 137.148,A -85,B 0,C 180,E1 -8256.037,E2 -8256.037} C_VEL
LIN {X 0,Y 459.988,Z 263.498,A -85,B 0,C 180,E1 -8258.341,E2 -8258.341} C_VEL
LIN {X 0,Y 459.621,Z 285.247,A -85,B 0,C 180,E1 -8258.78,E2 -8258.78} C_VEL
LIN {X 0,Y 459.198,Z 300.216,A -85,B 0,C 180,E1 -8259.253,E2 -8259.253} C_VEL
LIN {X 0,Y 458.594,Z 314.869,A -85,B 0,C 180,E1 -8259.888,E2 -8259.888} C_VEL
LIN {X 0,Y 457.85,Z 329.826,A -85,B 0,C 180,E1 -8260.729,E2 -8260.729} C_VEL
LIN {X 0,Y 457.037,Z 344.121,A -85,B 0,C 180,E1 -8261.741,E2 -8261.741} C_VEL
LIN {X 0,Y 456.333,Z 357.148,A -85,B 0,C 180,E1 -8262.873,E2 -8262.873} C_VEL
LIN {X 0,Y 455.555,Z 368.983,A -85,B 0,C 180,E1 -8264.107,E2 -8264.107} C_VEL
LIN {X 0,Y 454.889,Z 379.857,A -85,B 0,C 180,E1 -8265.459,E2 -8265.459} C_VEL
LIN {X 0,Y 454.221,Z 390.073,A -85,B 0,C 180,E1 -8266.975,E2 -8266.975} C_VEL
LIN {X 0,Y 453.757,Z 399.192,A -85,B 0,C 180,E1 -8268.61,E2 -8268.61} C_VEL
LIN {X 0,Y 453.298,Z 406.451,A -85,B 0,C 180,E1 -8270.18,E2 -8270.18} C_VEL
LIN {X 0,Y 452.995,Z 413.159,A -85,B 0,C 180,E1 -8271.973,E2 -8271.973} C_VEL
LIN {X 0,Y 452.811,Z 418.365,A -85,B 0,C 180,E1 -8273.762,E2 -8273.762} C_VEL
LIN {X 0,Y 452.631,Z 422.217,A -85,B 0,C 180,E1 -8275.547,E2 -8275.547} C_VEL
LIN {X 0,Y 452.632,Z 424.804,A -85,B 0,C 180,E1 -8277.33,E2 -8277.33} C_VEL
LIN {X 0,Y 452.498,Z 426.187,A -85,B 0,C 180,E1 -8279.11,E2 -8279.11} C_VEL
LIN {X 0,Y 452.499,Z 426.333,A -85,B 0,C 180,E1 -8280.89,E2 -8280.89} C_VEL
LIN {X 0,Y 452.673,Z 425.279,A -85,B 0,C 180,E1 -8282.669,E2 -8282.669} C_VEL
LIN {X 0,Y 452.722,Z 423.032,A -85,B 0,C 180,E1 -8284.451,E2 -8284.451} C_VEL
LIN {X 0,Y 452.923,Z 419.526,A -85,B 0,C 180,E1 -8286.235,E2 -8286.235} C_VEL
LIN {X 0,Y 453.082,Z 414.689,A -85,B 0,C 180,E1 -8288.025,E2 -8288.025} C_VEL
LIN {X 0,Y 453.439,Z 408.373,A -85,B 0,C 180,E1 -8289.816,E2 -8289.816} C_VEL
LIN {X 0,Y 453.922,Z 400.403,A -85,B 0,C 180,E1 -8291.611,E2 -8291.611} C_VEL
LIN {X 0,Y 454.498,Z 391.512,A -85,B 0,C 180,E1 -8293.238,E2 -8293.238} C_VEL
LIN {X 0,Y 455.238,Z 381.48,A -85,B 0,C 180,E1 -8294.757,E2 -8294.757} C_VEL
LIN {X 0,Y 455.969,Z 370.824,A -85,B 0,C 180,E1 -8296.107,E2 -8296.107} C_VEL
LIN {X 0,Y 456.836,Z 358.496,A -85,B 0,C 180,E1 -8297.409,E2 -8297.409} C_VEL
LIN {X 0,Y 457.568,Z 346.496,A -85,B 0,C 180,E1 -8298.469,E2 -8298.469} C_VEL
LIN {X 0,Y 458.42,Z 332.546,A -85,B 0,C 180,E1 -8299.478,E2 -8299.478} C_VEL
LIN {X 0,Y 459.127,Z 318.073,A -85,B 0,C 180,E1 -8300.321,E2 -8300.321} C_VEL
LIN {X 0,Y 459.776,Z 303.323,A -85,B 0,C 180,E1 -8300.984,E2 -8300.984} C_VEL
LIN {X 0,Y 460.28,Z 287.735,A -85,B 0,C 180,E1 -8301.497,E2 -8301.497} C_VEL
LIN {X 0,Y 460.84,Z 262.752,A -85,B 0,C 180,E1 -8302.028,E2 -8302.028} C_VEL
LIN {X 0,Y 463.276,Z 181.124,A -85,B 0,C 180,E1 -8303.704,E2 -8303.704} C_VEL
LIN {X 0,Y 464.672,Z 141.025,A -85,B 0,C 180,E1 -8304.582,E2 -8304.582} C_VEL
LIN {X 0,Y 459.374,Z 129.782,A -85,B 0,C 180,E1 -8305.294,E2 -8305.294} C_VEL
LIN {X 0,Y 455.835,Z 123.044,A -85,B 0,C 180,E1 -8305.805,E2 -8305.805} C_VEL
LIN {X 0,Y 453.489,Z 114.624,A -85,B 0,C 180,E1 -8308.125,E2 -8308.125} C_VEL
LIN {X 0,Y 453.463,Z 114.627,A -85,B 0,C 180,E1 -8311.524,E2 -8311.524} C_VEL
LIN {X 0,Y 453.481,Z 114.624,A -85,B 0,C 180,E1 -8314.776,E2 -8314.776} C_VEL
LIN {X 0,Y 453.456,Z 114.626,A -85,B 0,C 180,E1 -8318.312,E2 -8318.312} C_VEL
LIN {X 0,Y 453.469,Z 114.624,A -85,B 0,C 180,E1 -8320.611,E2 -8320.611} C_VEL
LIN {X 0,Y 453.48,Z 114.623,A -85,B 0,C 180,E1 -8324.528,E2 -8324.528} C_VEL
LIN {X 0,Y 453.435,Z 114.628,A -85,B 0,C 180,E1 -8328.071,E2 -8328.071} C_VEL
LIN {X 0,Y 453.446,Z 114.63,A -85,B 0,C 180,E1 -8330.801,E2 -8330.801} C_VEL
LIN {X 0,Y 453.448,Z 114.63,A -85,B 0,C 180,E1 -8333.917,E2 -8333.917} C_VEL
LIN {X 0,Y 453.499,Z 114.787,A -85,B 0,C 180,E1 -8336.19,E2 -8336.19} C_VEL
LIN {X 0,Y 455.88,Z 122.541,A -85,B 0,C 180,E1 -8337.984,E2 -8337.984} C_VEL
LIN {X 0,Y 458.26,Z 131.578,A -85,B 0,C 180,E1 -8339.85,E2 -8339.85} C_VEL
LIN {X 0,Y 459.787,Z 139.108,A -85,B 0,C 180,E1 -8341.258,E2 -8341.258} C_VEL
LIN {X 0,Y 458.327,Z 155.922,A -85,B 0,C 180,E1 -8343.842,E2 -8343.842} C_VEL
LIN {X 0,Y 458.016,Z 159.855,A -85,B 0,C 180,E1 -8344.404,E2 -8344.404} C_VEL
LIN {X 0,Y 461.584,Z 177.827,A -85,B 0,C 180,E1 -8345.137,E2 -8345.137} C_VEL
LIN {X 0,Y 463.611,Z 193.162,A -85,B 0,C 180,E1 -8345.654,E2 -8345.654} C_VEL
LIN {X 0,Y 460.975,Z 281.046,A -85,B 0,C 180,E1 -8347.477,E2 -8347.477} C_VEL
LIN {X 0,Y 459.859,Z 330.131,A -85,B 0,C 180,E1 -8348.453,E2 -8348.453} C_VEL
LIN {X 0,Y 458.946,Z 351.004,A -85,B 0,C 180,E1 -8349.085,E2 -8349.085} C_VEL
LIN {X 0,Y 458.36,Z 366.026,A -85,B 0,C 180,E1 -8349.702,E2 -8349.702} C_VEL
LIN {X 0,Y 457.544,Z 380.464,A -85,B 0,C 180,E1 -8350.483,E2 -8350.483} C_VEL
LIN {X 0,Y 456.821,Z 393.618,A -85,B 0,C 180,E1 -8351.384,E2 -8351.384} C_VEL
LIN {X 0,Y 456.011,Z 405.789,A -85,B 0,C 180,E1 -8352.395,E2 -8352.395} C_VEL
LIN {X 0,Y 455.115,Z 418.559,A -85,B 0,C 180,E1 -8353.682,E2 -8353.682} C_VEL
LIN {X 0,Y 454.46,Z 429.324,A -85,B 0,C 180,E1 -8354.987,E2 -8354.987} C_VEL
LIN {X 0,Y 453.865,Z 438.735,A -85,B 0,C 180,E1 -8356.341,E2 -8356.341} C_VEL
LIN {X 0,Y 453.344,Z 447.036,A -85,B 0,C 180,E1 -8357.752,E2 -8357.752} C_VEL
LIN {X 0,Y 453.051,Z 454.557,A -85,B 0,C 180,E1 -8359.272,E2 -8359.272} C_VEL
LIN {X 0,Y 452.712,Z 461.854,A -85,B 0,C 180,E1 -8361.069,E2 -8361.069} C_VEL
LIN {X 0,Y 452.643,Z 467.588,A -85,B 0,C 180,E1 -8362.865,E2 -8362.865} C_VEL
LIN {X 0,Y 452.54,Z 471.909,A -85,B 0,C 180,E1 -8364.653,E2 -8364.653} C_VEL
LIN {X 0,Y 452.491,Z 474.936,A -85,B 0,C 180,E1 -8366.438,E2 -8366.438} C_VEL
LIN {X 0,Y 452.509,Z 476.744,A -85,B 0,C 180,E1 -8368.22,E2 -8368.22} C_VEL
LIN {X 0,Y 452.44,Z 477.36,A -85,B 0,C 180,E1 -8370,E2 -8370} C_VEL
LIN {X 0,Y 452.508,Z 476.757,A -85,B 0,C 180,E1 -8371.78,E2 -8371.78} C_VEL
LIN {X 0,Y 452.503,Z 474.957,A -85,B 0,C 180,E1 -8373.562,E2 -8373.562} C_VEL
LIN {X 0,Y 452.543,Z 471.929,A -85,B 0,C 180,E1 -8375.347,E2 -8375.347} C_VEL
LIN {X 0,Y 452.644,Z 467.603,A -85,B 0,C 180,E1 -8377.135,E2 -8377.135} C_VEL
LIN {X 0,Y 452.709,Z 461.868,A -85,B 0,C 180,E1 -8378.931,E2 -8378.931} C_VEL
LIN {X 0,Y 453.058,Z 454.568,A -85,B 0,C 180,E1 -8380.728,E2 -8380.728} C_VEL
LIN {X 0,Y 453.374,Z 446.074,A -85,B 0,C 180,E1 -8382.421,E2 -8382.421} C_VEL
LIN {X 0,Y 453.904,Z 437.188,A -85,B 0,C 180,E1 -8383.886,E2 -8383.886} C_VEL
LIN {X 0,Y 454.521,Z 427.452,A -85,B 0,C 180,E1 -8385.24,E2 -8385.24} C_VEL
LIN {X 0,Y 455.175,Z 416.78,A -85,B 0,C 180,E1 -8386.494,E2 -8386.494} C_VEL
LIN {X 0,Y 455.973,Z 404.224,A -85,B 0,C 180,E1 -8387.723,E2 -8387.723} C_VEL
LIN {X 0,Y 456.839,Z 391.699,A -85,B 0,C 180,E1 -8388.732,E2 -8388.732} C_VEL
LIN {X 0,Y 457.614,Z 378.003,A -85,B 0,C 180,E1 -8389.631,E2 -8389.631} C_VEL
LIN {X 0,Y 458.374,Z 363.934,A -85,B 0,C 180,E1 -8390.356,E2 -8390.356} C_VEL
LIN {X 0,Y 458.92,Z 349.026,A -85,B 0,C 180,E1 -8390.936,E2 -8390.936} C_VEL
LIN {X 0,Y 459.461,Z 330.637,A -85,B 0,C 180,E1 -8391.444,E2 -8391.444} C_VEL
LIN {X 0,Y 461.344,Z 236.058,A -85,B 0,C 180,E1 -8393.185,E2 -8393.185} C_VEL
LIN {X 0,Y 462.808,Z 187.894,A -85,B 0,C 180,E1 -8394.219,E2 -8394.219} C_VEL
LIN {X 0,Y 459.371,Z 161.088,A -85,B 0,C 180,E1 -8395.138,E2 -8395.138} C_VEL
LIN {X 0,Y 459.055,Z 158.253,A -85,B 0,C 180,E1 -8395.25,E2 -8395.25} C_VEL
LIN {X 0,Y 460.124,Z 139.836,A -85,B 0,C 180,E1 -8397.273,E2 -8397.273} C_VEL
LIN {X 0,Y 458.582,Z 133.111,A -85,B 0,C 180,E1 -8398.125,E2 -8398.125} C_VEL
LIN {X 0,Y 453.483,Z 114.624,A -85,B 0,C 180,E1 -8400.592,E2 -8400.592} C_VEL
LIN {X 0,Y 453.465,Z 114.623,A -85,B 0,C 180,E1 -8403.914,E2 -8403.914} C_VEL
LIN {X 0,Y 453.448,Z 114.627,A -85,B 0,C 180,E1 -8407.19,E2 -8407.19} C_VEL
LIN {X 0,Y 453.469,Z 114.624,A -85,B 0,C 180,E1 -8410.612,E2 -8410.612} C_VEL
LIN {X 0,Y 453.48,Z 114.621,A -85,B 0,C 180,E1 -8414.529,E2 -8414.529} C_VEL
LIN {X 0,Y 453.435,Z 114.626,A -85,B 0,C 180,E1 -8418.071,E2 -8418.071} C_VEL
LIN {X 0,Y 453.447,Z 114.627,A -85,B 0,C 180,E1 -8420.801,E2 -8420.801} C_VEL
LIN {X 0,Y 453.45,Z 114.627,A -85,B 0,C 180,E1 -8423.917,E2 -8423.917} C_VEL
LIN {X 0,Y 453.474,Z 114.623,A -85,B 0,C 180,E1 -8427.151,E2 -8427.151} C_VEL
LIN {X 0,Y 453.462,Z 114.628,A -85,B 0,C 180,E1 -8430.268,E2 -8430.268} C_VEL
LIN {X 0,Y 453.467,Z 114.708,A -85,B 0,C 180,E1 -8433.261,E2 -8433.261} C_VEL
LIN {X 0,Y 455.465,Z 120.538,A -85,B 0,C 180,E1 -8434.278,E2 -8434.278} C_VEL
LIN {X 0,Y 461.122,Z 131.905,A -85,B 0,C 180,E1 -8435.062,E2 -8435.062} C_VEL
LIN {X 0,Y 464.611,Z 139.883,A -85,B 0,C 180,E1 -8435.534,E2 -8435.534} C_VEL
LIN {X 0,Y 461.554,Z 231.879,A -85,B 0,C 180,E1 -8437.478,E2 -8437.478} C_VEL
LIN {X 0,Y 460.271,Z 285.35,A -85,B 0,C 180,E1 -8438.555,E2 -8438.555} C_VEL
LIN {X 0,Y 459.771,Z 300.768,A -85,B 0,C 180,E1 -8439.032,E2 -8439.032} C_VEL
LIN {X 0,Y 459.182,Z 315.813,A -85,B 0,C 180,E1 -8439.681,E2 -8439.681} C_VEL
LIN {X 0,Y 458.534,Z 328.911,A -85,B 0,C 180,E1 -8440.411,E2 -8440.411} C_VEL
LIN {X 0,Y 457.822,Z 342.054,A -85,B 0,C 180,E1 -8441.31,E2 -8441.31} C_VEL
LIN {X 0,Y 456.976,Z 355.203,A -85,B 0,C 180,E1 -8442.403,E2 -8442.403} C_VEL
LIN {X 0,Y 456.057,Z 367.762,A -85,B 0,C 180,E1 -8443.666,E2 -8443.666} C_VEL
LIN {X 0,Y 455.377,Z 378.891,A -85,B 0,C 180,E1 -8445.019,E2 -8445.019} C_VEL
LIN {X 0,Y 454.62,Z 389.695,A -85,B 0,C 180,E1 -8446.592,E2 -8446.592} C_VEL
LIN {X 0,Y 454.092,Z 397.404,A -85,B 0,C 180,E1 -8447.94,E2 -8447.94} C_VEL
LIN {X 0,Y 453.626,Z 403.979,A -85,B 0,C 180,E1 -8449.286,E2 -8449.286} C_VEL
LIN {X 0,Y 453.246,Z 411.189,A -85,B 0,C 180,E1 -8451.08,E2 -8451.08} C_VEL
LIN {X 0,Y 452.94,Z 416.843,A -85,B 0,C 180,E1 -8452.87,E2 -8452.87} C_VEL
LIN {X 0,Y 452.905,Z 419.127,A -85,B 0,C 180,E1 -8453.764,E2 -8453.764} C_VEL
LIN {X 0,Y 452.686,Z 422.709,A -85,B 0,C 180,E1 -8455.548,E2 -8455.548} C_VEL
LIN {X 0,Y 452.669,Z 425.029,A -85,B 0,C 180,E1 -8457.331,E2 -8457.331} C_VEL
LIN {X 0,Y 452.497,Z 426.155,A -85,B 0,C 180,E1 -8459.11,E2 -8459.11} C_VEL
LIN {X 0,Y 452.497,Z 426.058,A -85,B 0,C 180,E1 -8460.89,E2 -8460.89} C_VEL
LIN {X 0,Y 452.618,Z 424.739,A -85,B 0,C 180,E1 -8462.67,E2 -8462.67} C_VEL
LIN {X 0,Y 452.612,Z 422.22,A -85,B 0,C 180,E1 -8464.453,E2 -8464.453} C_VEL
LIN {X 0,Y 452.816,Z 418.428,A -85,B 0,C 180,E1 -8466.237,E2 -8466.237} C_VEL
LIN {X 0,Y 452.984,Z 413.289,A -85,B 0,C 180,E1 -8468.027,E2 -8468.027} C_VEL
LIN {X 0,Y 453.263,Z 406.662,A -85,B 0,C 180,E1 -8469.821,E2 -8469.821} C_VEL
LIN {X 0,Y 453.702,Z 399.472,A -85,B 0,C 180,E1 -8471.391,E2 -8471.391} C_VEL
LIN {X 0,Y 454.119,Z 390.615,A -85,B 0,C 180,E1 -8472.997,E2 -8472.997} C_VEL
LIN {X 0,Y 454.803,Z 380.304,A -85,B 0,C 180,E1 -8474.543,E2 -8474.543} C_VEL
LIN {X 0,Y 455.465,Z 369.525,A -85,B 0,C 180,E1 -8475.896,E2 -8475.896} C_VEL
LIN {X 0,Y 456.212,Z 357.674,A -85,B 0,C 180,E1 -8477.144,E2 -8477.144} C_VEL
LIN {X 0,Y 457.04,Z 344.945,A -85,B 0,C 180,E1 -8478.259,E2 -8478.259} C_VEL
LIN {X 0,Y 457.754,Z 330.876,A -85,B 0,C 180,E1 -8479.275,E2 -8479.275} C_VEL
LIN {X 0,Y 458.523,Z 316.224,A -85,B 0,C 180,E1 -8480.116,E2 -8480.116} C_VEL
LIN {X 0,Y 459.057,Z 301.735,A -85,B 0,C 180,E1 -8480.764,E2 -8480.764} C_VEL
LIN {X 0,Y 459.541,Z 286.697,A -85,B 0,C 180,E1 -8481.257,E2 -8481.257} C_VEL
LIN {X 0,Y 459.829,Z 270.516,A -85,B 0,C 180,E1 -8481.608,E2 -8481.608} C_VEL
LIN {X 0,Y 462.363,Z 137.91,A -85,B 0,C 180,E1 -8484.014,E2 -8484.014} C_VEL
LIN {X 0,Y 453.669,Z 115.435,A -85,B 0,C 180,E1 -8484.917,E2 -8484.917} C_VEL
LIN {X 0,Y 453.519,Z 114.62,A -85,B 0,C 180,E1 -8485.101,E2 -8485.101} C_VEL
LIN {X 0,Y 453.468,Z 114.622,A -85,B 0,C 180,E1 -8488.715,E2 -8488.715} C_VEL
LIN {X 0,Y 453.463,Z 114.627,A -85,B 0,C 180,E1 -8491.8,E2 -8491.8} C_VEL
LIN {X 0,Y 453.477,Z 114.621,A -85,B 0,C 180,E1 -8494.99,E2 -8494.99} C_VEL
LIN {X 0,Y 453.459,Z 114.622,A -85,B 0,C 180,E1 -8498.313,E2 -8498.313} C_VEL
LIN {X 0,Y 453.472,Z 114.621,A -85,B 0,C 180,E1 -8500.612,E2 -8500.612} C_VEL
LIN {X 0,Y 453.461,Z 114.618,A -85,B 0,C 180,E1 -8504.222,E2 -8504.222} C_VEL
LIN {X 0,Y 453.423,Z 114.613,A -85,B 0,C 180,E1 -8507,E2 -8507} C_VEL
LIN {X 0,Y 453.472,Z 114.625,A -85,B 0,C 180,E1 -8509.413,E2 -8509.413} C_VEL
LIN {X 0,Y 453.452,Z 114.624,A -85,B 0,C 180,E1 -8512.81,E2 -8512.81} C_VEL
LIN {X 0,Y 453.469,Z 114.617,A -85,B 0,C 180,E1 -8516.087,E2 -8516.087} C_VEL
LIN {X 0,Y 453.457,Z 114.62,A -85,B 0,C 180,E1 -8519.239,E2 -8519.239} C_VEL
LIN {X 0,Y 453.462,Z 114.619,A -85,B 0,C 180,E1 -8521.739,E2 -8521.739} C_VEL
LIN {X 0,Y 452.807,Z 114.705,A -85,B 0,C 180,E1 -8522.48,E2 -8522.48} C_VEL
LIN {X 0,Y 449.935,Z 115.062,A -85,B 0,C 180,E1 -8523.683,E2 -8523.683} C_VEL
LIN {X 0,Y 447.509,Z 115.366,A -85,B 0,C 180,E1 -8524.654,E2 -8524.654} C_VEL
LIN {X 0,Y 446.486,Z 115.484,A -85,B 0,C 180,E1 -8525.405,E2 -8525.405} C_VEL
LIN {X 0,Y 446.413,Z 115.492,A -85,B 0,C 180,E1 -8525.659,E2 -8525.659} C_VEL
LIN {X 0,Y 446.451,Z 115.498,A -85,B 0,C 180,E1 -8528.773,E2 -8528.773} C_VEL
LIN {X 0,Y 446.442,Z 115.497,A -85,B 0,C 180,E1 -8531.649,E2 -8531.649} C_VEL
LIN {X 0,Y 446.461,Z 115.495,A -85,B 0,C 180,E1 -8534.478,E2 -8534.478} C_VEL
LIN {X 0,Y 446.52,Z 115.486,A -85,B 0,C 180,E1 -8537.384,E2 -8537.384} C_VEL
LIN {X 0,Y 446.515,Z 115.489,A -85,B 0,C 180,E1 -8540.944,E2 -8540.944} C_VEL
LIN {X 0,Y 446.602,Z 115.479,A -85,B 0,C 180,E1 -8543.676,E2 -8543.676} C_VEL
LIN {X 0,Y 446.657,Z 115.504,A -85,B 0,C 180,E1 -8547.633,E2 -8547.633} C_VEL
LIN {X 0,Y 450.279,Z 130.964,A -85,B 0,C 180,E1 -8550.135,E2 -8550.135} C_VEL
LIN {X 0,Y 451.418,Z 137.165,A -85,B 0,C 180,E1 -8551.115,E2 -8551.115} C_VEL
LIN {X 0,Y 451.198,Z 142.401,A -85,B 0,C 180,E1 -8551.869,E2 -8551.869} C_VEL
LIN {X 0,Y 456.321,Z 166.579,A -85,B 0,C 180,E1 -8552.593,E2 -8552.593} C_VEL
LIN {X 0,Y 454.248,Z 308.444,A -85,B 0,C 180,E1 -8554.909,E2 -8554.909} C_VEL
LIN {X 0,Y 453.793,Z 323.847,A -85,B 0,C 180,E1 -8555.332,E2 -8555.332} C_VEL
LIN {X 0,Y 453.166,Z 338.22,A -85,B 0,C 180,E1 -8555.897,E2 -8555.897} C_VEL
LIN {X 0,Y 452.437,Z 351.457,A -85,B 0,C 180,E1 -8556.578,E2 -8556.578} C_VEL
LIN {X 0,Y 451.53,Z 365.492,A -85,B 0,C 180,E1 -8557.49,E2 -8557.49} C_VEL
LIN {X 0,Y 450.593,Z 378.336,A -85,B 0,C 180,E1 -8558.521,E2 -8558.521} C_VEL
LIN {X 0,Y 449.611,Z 391.015,A -85,B 0,C 180,E1 -8559.758,E2 -8559.758} C_VEL
LIN {X 0,Y 448.72,Z 402.162,A -85,B 0,C 180,E1 -8561.062,E2 -8561.062} C_VEL
LIN {X 0,Y 447.869,Z 412.223,A -85,B 0,C 180,E1 -8562.461,E2 -8562.461} C_VEL
LIN {X 0,Y 447.113,Z 422.054,A -85,B 0,C 180,E1 -8564.101,E2 -8564.101} C_VEL
LIN {X 0,Y 446.485,Z 430.635,A -85,B 0,C 180,E1 -8565.845,E2 -8565.845} C_VEL
LIN {X 0,Y 446.086,Z 437.011,A -85,B 0,C 180,E1 -8567.418,E2 -8567.418} C_VEL
LIN {X 0,Y 445.714,Z 443.244,A -85,B 0,C 180,E1 -8569.337,E2 -8569.337} C_VEL
LIN {X 0,Y 445.518,Z 447.978,A -85,B 0,C 180,E1 -8571.274,E2 -8571.274} C_VEL
LIN {X 0,Y 445.282,Z 451.33,A -85,B 0,C 180,E1 -8573.24,E2 -8573.24} C_VEL
LIN {X 0,Y 445.199,Z 453.297,A -85,B 0,C 180,E1 -8575.228,E2 -8575.228} C_VEL
LIN {X 0,Y 445.222,Z 453.879,A -85,B 0,C 180,E1 -8577.244,E2 -8577.244} C_VEL
LIN {X 0,Y 445.265,Z 453.021,A -85,B 0,C 180,E1 -8579.295,E2 -8579.295} C_VEL
LIN {X 0,Y 445.362,Z 450.634,A -85,B 0,C 180,E1 -8581.383,E2 -8581.383} C_VEL
LIN {X 0,Y 445.52,Z 447.12,A -85,B 0,C 180,E1 -8583.272,E2 -8583.272} C_VEL
LIN {X 0,Y 445.756,Z 442.928,A -85,B 0,C 180,E1 -8584.929,E2 -8584.929} C_VEL
LIN {X 0,Y 446.086,Z 436.878,A -85,B 0,C 180,E1 -8586.776,E2 -8586.776} C_VEL
LIN {X 0,Y 446.595,Z 429.8,A -85,B 0,C 180,E1 -8588.502,E2 -8588.502} C_VEL
LIN {X 0,Y 447.16,Z 421.74,A -85,B 0,C 180,E1 -8590.12,E2 -8590.12} C_VEL
LIN {X 0,Y 447.844,Z 413.336,A -85,B 0,C 180,E1 -8591.531,E2 -8591.531} C_VEL
LIN {X 0,Y 448.734,Z 402.984,A -85,B 0,C 180,E1 -8592.997,E2 -8592.997} C_VEL
LIN {X 0,Y 449.582,Z 392.143,A -85,B 0,C 180,E1 -8594.287,E2 -8594.287} C_VEL
LIN {X 0,Y 450.572,Z 380.79,A -85,B 0,C 180,E1 -8595.419,E2 -8595.419} C_VEL
LIN {X 0,Y 451.55,Z 367.484,A -85,B 0,C 180,E1 -8596.525,E2 -8596.525} C_VEL
LIN {X 0,Y 452.477,Z 353.577,A -85,B 0,C 180,E1 -8597.461,E2 -8597.461} C_VEL
LIN {X 0,Y 453.241,Z 340.053,A -85,B 0,C 180,E1 -8598.182,E2 -8598.182} C_VEL
LIN {X 0,Y 453.944,Z 324.412,A -85,B 0,C 180,E1 -8598.813,E2 -8598.813} C_VEL
LIN {X 0,Y 454.432,Z 309.394,A -85,B 0,C 180,E1 -8599.229,E2 -8599.229} C_VEL
LIN {X 0,Y 456.687,Z 161.785,A -85,B 0,C 180,E1 -8601.66,E2 -8601.66} C_VEL
LIN {X 0,Y 452.878,Z 141.166,A -85,B 0,C 180,E1 -8602.256,E2 -8602.256} C_VEL
LIN {X 0,Y 452.479,Z 137.373,A -85,B 0,C 180,E1 -8602.716,E2 -8602.716} C_VEL
LIN {X 0,Y 448.719,Z 123.17,A -85,B 0,C 180,E1 -8604.584,E2 -8604.584} C_VEL
LIN {X 0,Y 446.476,Z 115.497,A -85,B 0,C 180,E1 -8605.652,E2 -8605.652} C_VEL
LIN {X 0,Y 446.419,Z 115.501,A -85,B 0,C 180,E1 -8608.699,E2 -8608.699} C_VEL
LIN {X 0,Y 446.487,Z 115.496,A -85,B 0,C 180,E1 -8611.821,E2 -8611.821} C_VEL
LIN {X 0,Y 446.486,Z 115.496,A -85,B 0,C 180,E1 -8614.755,E2 -8614.755} C_VEL
LIN {X 0,Y 448.45,Z 120.574,A -85,B 0,C 180,E1 -8614.982,E2 -8614.982} C_VEL
LIN {X 0,Y 455.786,Z 138.902,A -85,B 0,C 180,E1 -8615.738,E2 -8615.738} C_VEL
LIN {X 0,Y 453.131,Z 271.848,A -85,B 0,C 180,E1 -8618.218,E2 -8618.218} C_VEL
LIN {X 0,Y 452.755,Z 288.782,A -85,B 0,C 180,E1 -8618.603,E2 -8618.603} C_VEL
LIN {X 0,Y 452.271,Z 303.643,A -85,B 0,C 180,E1 -8619.118,E2 -8619.118} C_VEL
LIN {X 0,Y 451.589,Z 319.402,A -85,B 0,C 180,E1 -8619.859,E2 -8619.859} C_VEL
LIN {X 0,Y 450.91,Z 332.613,A -85,B 0,C 180,E1 -8620.658,E2 -8620.658} C_VEL
LIN {X 0,Y 450.1,Z 346.467,A -85,B 0,C 180,E1 -8621.685,E2 -8621.685} C_VEL
LIN {X 0,Y 449.332,Z 359.122,A -85,B 0,C 180,E1 -8622.829,E2 -8622.829} C_VEL
LIN {X 0,Y 448.543,Z 370.744,A -85,B 0,C 180,E1 -8624.085,E2 -8624.085} C_VEL
LIN {X 0,Y 447.822,Z 381.409,A -85,B 0,C 180,E1 -8625.457,E2 -8625.457} C_VEL
LIN {X 0,Y 447.235,Z 390.351,A -85,B 0,C 180,E1 -8626.816,E2 -8626.816} C_VEL
LIN {X 0,Y 446.757,Z 399.271,A -85,B 0,C 180,E1 -8628.429,E2 -8628.429} C_VEL
LIN {X 0,Y 446.28,Z 406.602,A -85,B 0,C 180,E1 -8630.024,E2 -8630.024} C_VEL
LIN {X 0,Y 445.947,Z 413.376,A -85,B 0,C 180,E1 -8631.846,E2 -8631.846} C_VEL
LIN {X 0,Y 445.745,Z 418.64,A -85,B 0,C 180,E1 -8633.663,E2 -8633.663} C_VEL
LIN {X 0,Y 445.546,Z 422.539,A -85,B 0,C 180,E1 -8635.476,E2 -8635.476} C_VEL
LIN {X 0,Y 445.555,Z 425.167,A -85,B 0,C 180,E1 -8637.287,E2 -8637.287} C_VEL
LIN {X 0,Y 445.435,Z 426.575,A -85,B 0,C 180,E1 -8639.096,E2 -8639.096} C_VEL
LIN {X 0,Y 445.437,Z 426.751,A -85,B 0,C 180,E1 -8640.904,E2 -8640.904} C_VEL
LIN {X 0,Y 445.593,Z 425.726,A -85,B 0,C 180,E1 -8642.712,E2 -8642.712} C_VEL
LIN {X 0,Y 445.641,Z 423.501,A -85,B 0,C 180,E1 -8644.522,E2 -8644.522} C_VEL
LIN {X 0,Y 445.882,Z 420.008,A -85,B 0,C 180,E1 -8646.334,E2 -8646.334} C_VEL
LIN {X 0,Y 446.046,Z 415.191,A -85,B 0,C 180,E1 -8648.152,E2 -8648.152} C_VEL
LIN {X 0,Y 446.444,Z 408.892,A -85,B 0,C 180,E1 -8649.972,E2 -8649.972} C_VEL
LIN {X 0,Y 446.968,Z 400.933,A -85,B 0,C 180,E1 -8651.795,E2 -8651.795} C_VEL
LIN {X 0,Y 447.579,Z 392.161,A -85,B 0,C 180,E1 -8653.431,E2 -8653.431} C_VEL
LIN {X 0,Y 448.373,Z 382.049,A -85,B 0,C 180,E1 -8654.988,E2 -8654.988} C_VEL
LIN {X 0,Y 449.159,Z 371.431,A -85,B 0,C 180,E1 -8656.358,E2 -8656.358} C_VEL
LIN {X 0,Y 450.086,Z 359.349,A -85,B 0,C 180,E1 -8657.657,E2 -8657.657} C_VEL
LIN {X 0,Y 450.873,Z 347.2,A -85,B 0,C 180,E1 -8658.753,E2 -8658.753} C_VEL
LIN {X 0,Y 451.786,Z 333.343,A -85,B 0,C 180,E1 -8659.776,E2 -8659.776} C_VEL
LIN {X 0,Y 452.541,Z 319.008,A -85,B 0,C 180,E1 -8660.63,E2 -8660.63} C_VEL
LIN {X 0,Y 453.263,Z 303.853,A -85,B 0,C 180,E1 -8661.327,E2 -8661.327} C_VEL
LIN {X 0,Y 453.785,Z 288.356,A -85,B 0,C 180,E1 -8661.85,E2 -8661.85} C_VEL
LIN {X 0,Y 454.455,Z 262.521,A -85,B 0,C 180,E1 -8662.414,E2 -8662.414} C_VEL
LIN {X 0,Y 457.01,Z 183.479,A -85,B 0,C 180,E1 -8664.096,E2 -8664.096} C_VEL
LIN {X 0,Y 458.618,Z 143.199,A -85,B 0,C 180,E1 -8665.004,E2 -8665.004} C_VEL
LIN {X 0,Y 453.073,Z 131.739,A -85,B 0,C 180,E1 -8665.787,E2 -8665.787} C_VEL
LIN {X 0,Y 448.906,Z 123.984,A -85,B 0,C 180,E1 -8666.404,E2 -8666.404} C_VEL
LIN {X 0,Y 446.423,Z 115.504,A -85,B 0,C 180,E1 -8668.888,E2 -8668.888} C_VEL
LIN {X 0,Y 446.415,Z 115.506,A -85,B 0,C 180,E1 -8671.774,E2 -8671.774} C_VEL
LIN {X 0,Y 446.421,Z 115.503,A -85,B 0,C 180,E1 -8674.523,E2 -8674.523} C_VEL
LIN {X 0,Y 446.41,Z 115.504,A -85,B 0,C 180,E1 -8678.078,E2 -8678.078} C_VEL
LIN {X 0,Y 446.399,Z 115.506,A -85,B 0,C 180,E1 -8681.394,E2 -8681.394} C_VEL
LIN {X 0,Y 446.448,Z 115.5,A -85,B 0,C 180,E1 -8685.104,E2 -8685.104} C_VEL
LIN {X 0,Y 446.399,Z 115.506,A -85,B 0,C 180,E1 -8688.606,E2 -8688.606} C_VEL
LIN {X 0,Y 446.409,Z 115.505,A -85,B 0,C 180,E1 -8691.922,E2 -8691.922} C_VEL
LIN {X 0,Y 446.444,Z 115.537,A -85,B 0,C 180,E1 -8695.412,E2 -8695.412} C_VEL
LIN {X 0,Y 449.58,Z 125.7,A -85,B 0,C 180,E1 -8697.893,E2 -8697.893} C_VEL
LIN {X 0,Y 452.047,Z 135.269,A -85,B 0,C 180,E1 -8699.912,E2 -8699.912} C_VEL
LIN {X 0,Y 453.192,Z 141.388,A -85,B 0,C 180,E1 -8701.08,E2 -8701.08} C_VEL
LIN {X 0,Y 451.51,Z 158.957,A -85,B 0,C 180,E1 -8703.836,E2 -8703.836} C_VEL
LIN {X 0,Y 455.238,Z 177.563,A -85,B 0,C 180,E1 -8704.644,E2 -8704.644} C_VEL
LIN {X 0,Y 457.434,Z 193.972,A -85,B 0,C 180,E1 -8705.231,E2 -8705.231} C_VEL
LIN {X 0,Y 454.533,Z 281.661,A -85,B 0,C 180,E1 -8707.11,E2 -8707.11} C_VEL
LIN {X 0,Y 453.335,Z 329.638,A -85,B 0,C 180,E1 -8708.097,E2 -8708.097} C_VEL
LIN {X 0,Y 452.346,Z 350.362,A -85,B 0,C 180,E1 -8708.74,E2 -8708.74} C_VEL
LIN {X 0,Y 451.67,Z 365.982,A -85,B 0,C 180,E1 -8709.387,E2 -8709.387} C_VEL
LIN {X 0,Y 450.834,Z 380.384,A -85,B 0,C 180,E1 -8710.18,E2 -8710.18} C_VEL
LIN {X 0,Y 450.077,Z 393.514,A -85,B 0,C 180,E1 -8711.094,E2 -8711.094} C_VEL
LIN {X 0,Y 449.176,Z 405.671,A -85,B 0,C 180,E1 -8712.118,E2 -8712.118} C_VEL
LIN {X 0,Y 448.358,Z 417.177,A -85,B 0,C 180,E1 -8713.287,E2 -8713.287} C_VEL
LIN {X 0,Y 447.531,Z 429.168,A -85,B 0,C 180,E1 -8714.749,E2 -8714.749} C_VEL
LIN {X 0,Y 446.886,Z 438.569,A -85,B 0,C 180,E1 -8716.123,E2 -8716.123} C_VEL
LIN {X 0,Y 446.306,Z 447.434,A -85,B 0,C 180,E1 -8717.662,E2 -8717.662} C_VEL
LIN {X 0,Y 445.97,Z 455.402,A -85,B 0,C 180,E1 -8719.329,E2 -8719.329} C_VEL
LIN {X 0,Y 445.635,Z 461.677,A -85,B 0,C 180,E1 -8720.926,E2 -8720.926} C_VEL
LIN {X 0,Y 445.565,Z 467.408,A -85,B 0,C 180,E1 -8722.751,E2 -8722.751} C_VEL
LIN {X 0,Y 445.439,Z 471.727,A -85,B 0,C 180,E1 -8724.568,E2 -8724.568} C_VEL
LIN {X 0,Y 445.388,Z 474.753,A -85,B 0,C 180,E1 -8726.381,E2 -8726.381} C_VEL
LIN {X 0,Y 445.424,Z 476.56,A -85,B 0,C 180,E1 -8728.192,E2 -8728.192} C_VEL
LIN {X 0,Y 445.348,Z 477.175,A -85,B 0,C 180,E1 -8730,E2 -8730} C_VEL
LIN {X 0,Y 445.422,Z 476.57,A -85,B 0,C 180,E1 -8731.808,E2 -8731.808} C_VEL
LIN {X 0,Y 445.399,Z 474.766,A -85,B 0,C 180,E1 -8733.619,E2 -8733.619} C_VEL
LIN {X 0,Y 445.46,Z 471.735,A -85,B 0,C 180,E1 -8735.432,E2 -8735.432} C_VEL
LIN {X 0,Y 445.565,Z 467.403,A -85,B 0,C 180,E1 -8737.249,E2 -8737.249} C_VEL
LIN {X 0,Y 445.632,Z 461.663,A -85,B 0,C 180,E1 -8739.074,E2 -8739.074} C_VEL
LIN {X 0,Y 445.999,Z 454.354,A -85,B 0,C 180,E1 -8740.9,E2 -8740.9} C_VEL
LIN {X 0,Y 446.32,Z 446.475,A -85,B 0,C 180,E1 -8742.504,E2 -8742.504} C_VEL
LIN {X 0,Y 446.931,Z 436.953,A -85,B 0,C 180,E1 -8744.107,E2 -8744.107} C_VEL
LIN {X 0,Y 447.607,Z 427.204,A -85,B 0,C 180,E1 -8745.481,E2 -8745.481} C_VEL
LIN {X 0,Y 448.244,Z 417.002,A -85,B 0,C 180,E1 -8746.704,E2 -8746.704} C_VEL
LIN {X 0,Y 449.058,Z 405.242,A -85,B 0,C 180,E1 -8747.887,E2 -8747.887} C_VEL
LIN {X 0,Y 449.972,Z 392.974,A -85,B 0,C 180,E1 -8748.91,E2 -8748.91} C_VEL
LIN {X 0,Y 450.793,Z 379.624,A -85,B 0,C 180,E1 -8749.821,E2 -8749.821} C_VEL
LIN {X 0,Y 451.634,Z 364.809,A -85,B 0,C 180,E1 -8750.614,E2 -8750.614} C_VEL
LIN {X 0,Y 452.217,Z 349.977,A -85,B 0,C 180,E1 -8751.212,E2 -8751.212} C_VEL
LIN {X 0,Y 452.69,Z 334.574,A -85,B 0,C 180,E1 -8751.636,E2 -8751.636} C_VEL
LIN {X 0,Y 453.95,Z 273.311,A -85,B 0,C 180,E1 -8752.801,E2 -8752.801} C_VEL
LIN {X 0,Y 456.651,Z 189.052,A -85,B 0,C 180,E1 -8754.635,E2 -8754.635} C_VEL
LIN {X 0,Y 453.35,Z 162.399,A -85,B 0,C 180,E1 -8755.586,E2 -8755.586} C_VEL
LIN {X 0,Y 452.44,Z 155.526,A -85,B 0,C 180,E1 -8755.881,E2 -8755.881} C_VEL
LIN {X 0,Y 453.326,Z 140.811,A -85,B 0,C 180,E1 -8757.526,E2 -8757.526} C_VEL
LIN {X 0,Y 447.438,Z 119.054,A -85,B 0,C 180,E1 -8760.422,E2 -8760.422} C_VEL
LIN {X 0,Y 446.448,Z 115.502,A -85,B 0,C 180,E1 -8760.935,E2 -8760.935} C_VEL
LIN {X 0,Y 446.423,Z 115.502,A -85,B 0,C 180,E1 -8763.449,E2 -8763.449} C_VEL
LIN {X 0,Y 446.399,Z 115.506,A -85,B 0,C 180,E1 -8766.746,E2 -8766.746} C_VEL
LIN {X 0,Y 446.4,Z 115.505,A -85,B 0,C 180,E1 -8769.517,E2 -8769.517} C_VEL
LIN {X 0,Y 446.375,Z 115.507,A -85,B 0,C 180,E1 -8772.611,E2 -8772.611} C_VEL
LIN {X 0,Y 446.448,Z 115.496,A -85,B 0,C 180,E1 -8775.104,E2 -8775.104} C_VEL
LIN {X 0,Y 446.399,Z 115.505,A -85,B 0,C 180,E1 -8778.606,E2 -8778.606} C_VEL
LIN {X 0,Y 446.409,Z 115.504,A -85,B 0,C 180,E1 -8781.922,E2 -8781.922} C_VEL
LIN {X 0,Y 446.421,Z 115.501,A -85,B 0,C 180,E1 -8785.477,E2 -8785.477} C_VEL
LIN {X 0,Y 446.413,Z 115.505,A -85,B 0,C 180,E1 -8788.7,E2 -8788.7} C_VEL
LIN {X 0,Y 446.446,Z 115.501,A -85,B 0,C 180,E1 -8791.831,E2 -8791.831} C_VEL
LIN {X 0,Y 446.47,Z 115.684,A -85,B 0,C 180,E1 -8792.649,E2 -8792.649} C_VEL
LIN {X 0,Y 448.419,Z 121.196,A -85,B 0,C 180,E1 -8793.655,E2 -8793.655} C_VEL
LIN {X 0,Y 454.339,Z 132.561,A -85,B 0,C 180,E1 -8794.514,E2 -8794.514} C_VEL
LIN {X 0,Y 458.516,Z 142.079,A -85,B 0,C 180,E1 -8795.115,E2 -8795.115} C_VEL
LIN {X 0,Y 455.248,Z 231.04,A -85,B 0,C 180,E1 -8797.058,E2 -8797.058} C_VEL
LIN {X 0,Y 453.787,Z 286.348,A -85,B 0,C 180,E1 -8798.213,E2 -8798.213} C_VEL
LIN {X 0,Y 453.233,Z 302.12,A -85,B 0,C 180,E1 -8798.72,E2 -8798.72} C_VEL
LIN {X 0,Y 452.585,Z 316.771,A -85,B 0,C 180,E1 -8799.372,E2 -8799.372} C_VEL
LIN {X 0,Y 451.914,Z 329.713,A -85,B 0,C 180,E1 -8800.112,E2 -8800.112} C_VEL
LIN {X 0,Y 451.143,Z 342.766,A -85,B 0,C 180,E1 -8801.023,E2 -8801.023} C_VEL
LIN {X 0,Y 450.245,Z 355.988,A -85,B 0,C 180,E1 -8802.145,E2 -8802.145} C_VEL
LIN {X 0,Y 449.259,Z 368.366,A -85,B 0,C 180,E1 -8803.412,E2 -8803.412} C_VEL
LIN {X 0,Y 448.536,Z 379.456,A -85,B 0,C 180,E1 -8804.785,E2 -8804.785} C_VEL
LIN {X 0,Y 447.713,Z 390.239,A -85,B 0,C 180,E1 -8806.381,E2 -8806.381} C_VEL
LIN {X 0,Y 447.062,Z 399.133,A -85,B 0,C 180,E1 -8807.978,E2 -8807.978} C_VEL
LIN {X 0,Y 446.565,Z 406.472,A -85,B 0,C 180,E1 -8809.573,E2 -8809.573} C_VEL
LIN {X 0,Y 446.148,Z 413.276,A -85,B 0,C 180,E1 -8811.394,E2 -8811.394} C_VEL
LIN {X 0,Y 445.855,Z 418.642,A -85,B 0,C 180,E1 -8813.25,E2 -8813.25} C_VEL
LIN {X 0,Y 445.634,Z 421.547,A -85,B 0,C 180,E1 -8814.571,E2 -8814.571} C_VEL
LIN {X 0,Y 445.632,Z 424.464,A -85,B 0,C 180,E1 -8816.383,E2 -8816.383} C_VEL
LIN {X 0,Y 445.523,Z 426.16,A -85,B 0,C 180,E1 -8818.192,E2 -8818.192} C_VEL
LIN {X 0,Y 445.411,Z 426.655,A -85,B 0,C 180,E1 -8820,E2 -8820} C_VEL
LIN {X 0,Y 445.474,Z 425.915,A -85,B 0,C 180,E1 -8821.808,E2 -8821.808} C_VEL
LIN {X 0,Y 445.612,Z 423.958,A -85,B 0,C 180,E1 -8823.617,E2 -8823.617} C_VEL
LIN {X 0,Y 445.629,Z 420.768,A -85,B 0,C 180,E1 -8825.43,E2 -8825.43} C_VEL
LIN {X 0,Y 445.787,Z 416.263,A -85,B 0,C 180,E1 -8827.246,E2 -8827.246} C_VEL
LIN {X 0,Y 446.064,Z 410.338,A -85,B 0,C 180,E1 -8829.065,E2 -8829.065} C_VEL
LIN {X 0,Y 446.439,Z 402.823,A -85,B 0,C 180,E1 -8830.889,E2 -8830.889} C_VEL
LIN {X 0,Y 446.861,Z 395.97,A -85,B 0,C 180,E1 -8832.259,E2 -8832.259} C_VEL
LIN {X 0,Y 447.432,Z 386.463,A -85,B 0,C 180,E1 -8833.86,E2 -8833.86} C_VEL
LIN {X 0,Y 448.093,Z 376.749,A -85,B 0,C 180,E1 -8835.231,E2 -8835.231} C_VEL
LIN {X 0,Y 448.885,Z 365.188,A -85,B 0,C 180,E1 -8836.603,E2 -8836.603} C_VEL
LIN {X 0,Y 449.655,Z 352.844,A -85,B 0,C 180,E1 -8837.828,E2 -8837.828} C_VEL
LIN {X 0,Y 450.416,Z 339.941,A -85,B 0,C 180,E1 -8838.891,E2 -8838.891} C_VEL
LIN {X 0,Y 451.187,Z 326.425,A -85,B 0,C 180,E1 -8839.804,E2 -8839.804} C_VEL
LIN {X 0,Y 451.928,Z 311.577,A -85,B 0,C 180,E1 -8840.601,E2 -8840.601} C_VEL
LIN {X 0,Y 452.453,Z 296.087,A -85,B 0,C 180,E1 -8841.235,E2 -8841.235} C_VEL
LIN {X 0,Y 452.884,Z 280.28,A -85,B 0,C 180,E1 -8841.686,E2 -8841.686} C_VEL
LIN {X 0,Y 455.743,Z 139.666,A -85,B 0,C 180,E1 -8844.315,E2 -8844.315} C_VEL
LIN {X 0,Y 446.522,Z 115.876,A -85,B 0,C 180,E1 -8845.276,E2 -8845.276} C_VEL
LIN {X 0,Y 446.473,Z 115.497,A -85,B 0,C 180,E1 -8845.401,E2 -8845.401} C_VEL
LIN {X 0,Y 446.44,Z 115.5,A -85,B 0,C 180,E1 -8848.182,E2 -8848.182} C_VEL
LIN {X 0,Y 446.416,Z 115.504,A -85,B 0,C 180,E1 -8851.301,E2 -8851.301} C_VEL
LIN {X 0,Y 446.423,Z 115.499,A -85,B 0,C 180,E1 -8854.524,E2 -8854.524} C_VEL
LIN {X 0,Y 446.412,Z 115.501,A -85,B 0,C 180,E1 -8858.079,E2 -8858.079} C_VEL
LIN {X 0,Y 446.403,Z 115.507,A -85,B 0,C 180,E1 -8861.394,E2 -8861.394} C_VEL
LIN {X 0,Y 446.452,Z 115.49,A -85,B 0,C 180,E1 -8865.104,E2 -8865.104} C_VEL
LIN {X 0,Y 446.402,Z 115.495,A -85,B 0,C 180,E1 -8868.606,E2 -8868.606} C_VEL
LIN {X 0,Y 446.412,Z 115.498,A -85,B 0,C 180,E1 -8871.922,E2 -8871.922} C_VEL
LIN {X 0,Y 446.425,Z 115.497,A -85,B 0,C 180,E1 -8875.477,E2 -8875.477} C_VEL
LIN {X 0,Y 446.41,Z 115.505,A -85,B 0,C 180,E1 -8878.699,E2 -8878.699} C_VEL
LIN {X 0,Y 446.428,Z 115.495,A -85,B 0,C 180,E1 -8881.836,E2 -8881.836} C_VEL
LIN {X 0,Y 446.424,Z 115.497,A -85,B 0,C 180,E1 -8884.846,E2 -8884.846} C_VEL
LIN {X 0,Y 446.413,Z 115.492,A -85,B 0,C 180,E1 -8885.659,E2 -8885.659} C_VEL
LIN {X 0,Y 445.775,Z 115.575,A -85,B 0,C 180,E1 -8886.413,E2 -8886.413} C_VEL
LIN {X 0,Y 442.93,Z 115.934,A -85,B 0,C 180,E1 -8887.637,E2 -8887.637} C_VEL
LIN {X 0,Y 440.505,Z 116.241,A -85,B 0,C 180,E1 -8888.625,E2 -8888.625} C_VEL
LIN {X 0,Y 439.462,Z 116.363,A -85,B 0,C 180,E1 -8889.388,E2 -8889.388} C_VEL
LIN {X 0,Y 439.377,Z 116.372,A -85,B 0,C 180,E1 -8889.647,E2 -8889.647} C_VEL
LIN {X 0,Y 439.391,Z 116.379,A -85,B 0,C 180,E1 -8892.308,E2 -8892.308} C_VEL
LIN {X 0,Y 439.401,Z 116.376,A -85,B 0,C 180,E1 -8895.172,E2 -8895.172} C_VEL
LIN {X 0,Y 439.487,Z 116.365,A -85,B 0,C 180,E1 -8898.001,E2 -8898.001} C_VEL
LIN {X 0,Y 439.484,Z 116.364,A -85,B 0,C 180,E1 -8901.725,E2 -8901.725} C_VEL
LIN {X 0,Y 439.595,Z 116.357,A -85,B 0,C 180,E1 -8904.495,E2 -8904.495} C_VEL
LIN {X 0,Y 439.645,Z 116.509,A -85,B 0,C 180,E1 -8907.309,E2 -8907.309} C_VEL
LIN {X 0,Y 443.231,Z 131.629,A -85,B 0,C 180,E1 -8909.787,E2 -8909.787} C_VEL
LIN {X 0,Y 444.619,Z 138.59,A -85,B 0,C 180,E1 -8910.906,E2 -8910.906} C_VEL
LIN {X 0,Y 444.527,Z 142.837,A -85,B 0,C 180,E1 -8911.5,E2 -8911.5} C_VEL
LIN {X 0,Y 449.814,Z 167.179,A -85,B 0,C 180,E1 -8912.239,E2 -8912.239} C_VEL
LIN {X 0,Y 447.65,Z 308.841,A -85,B 0,C 180,E1 -8914.587,E2 -8914.587} C_VEL
LIN {X 0,Y 447.153,Z 324.213,A -85,B 0,C 180,E1 -8915.016,E2 -8915.016} C_VEL
LIN {X 0,Y 446.52,Z 338.404,A -85,B 0,C 180,E1 -8915.583,E2 -8915.583} C_VEL
LIN {X 0,Y 445.685,Z 352.713,A -85,B 0,C 180,E1 -8916.337,E2 -8916.337} C_VEL
LIN {X 0,Y 444.745,Z 366.529,A -85,B 0,C 180,E1 -8917.263,E2 -8917.263} C_VEL
LIN {X 0,Y 443.75,Z 379.25,A -85,B 0,C 180,E1 -8918.309,E2 -8918.309} C_VEL
LIN {X 0,Y 442.767,Z 391.416,A -85,B 0,C 180,E1 -8919.521,E2 -8919.521} C_VEL
LIN {X 0,Y 441.894,Z 401.959,A -85,B 0,C 180,E1 -8920.77,E2 -8920.77} C_VEL
LIN {X 0,Y 440.976,Z 412.078,A -85,B 0,C 180,E1 -8922.191,E2 -8922.191} C_VEL
LIN {X 0,Y 440.159,Z 421.985,A -85,B 0,C 180,E1 -8923.857,E2 -8923.857} C_VEL
LIN {X 0,Y 439.526,Z 430.217,A -85,B 0,C 180,E1 -8925.535,E2 -8925.535} C_VEL
LIN {X 0,Y 439.066,Z 437.015,A -85,B 0,C 180,E1 -8927.225,E2 -8927.225} C_VEL
LIN {X 0,Y 438.683,Z 442.93,A -85,B 0,C 180,E1 -8929.051,E2 -8929.051} C_VEL
LIN {X 0,Y 438.493,Z 446.972,A -85,B 0,C 180,E1 -8930.647,E2 -8930.647} C_VEL
LIN {X 0,Y 438.239,Z 450.709,A -85,B 0,C 180,E1 -8932.637,E2 -8932.637} C_VEL
LIN {X 0,Y 438.107,Z 453.059,A -85,B 0,C 180,E1 -8934.651,E2 -8934.651} C_VEL
LIN {X 0,Y 438.104,Z 454.03,A -85,B 0,C 180,E1 -8936.691,E2 -8936.691} C_VEL
LIN {X 0,Y 438.13,Z 453.921,A -85,B 0,C 180,E1 -8938.084,E2 -8938.084} C_VEL
LIN {X 0,Y 438.219,Z 452.654,A -85,B 0,C 180,E1 -8939.998,E2 -8939.998} C_VEL
LIN {X 0,Y 438.329,Z 450.081,A -85,B 0,C 180,E1 -8941.945,E2 -8941.945} C_VEL
LIN {X 0,Y 438.509,Z 446.925,A -85,B 0,C 180,E1 -8943.549,E2 -8943.549} C_VEL
LIN {X 0,Y 438.755,Z 442.637,A -85,B 0,C 180,E1 -8945.222,E2 -8945.222} C_VEL
LIN {X 0,Y 439.115,Z 436.444,A -85,B 0,C 180,E1 -8947.103,E2 -8947.103} C_VEL
LIN {X 0,Y 439.676,Z 429.212,A -85,B 0,C 180,E1 -8948.858,E2 -8948.858} C_VEL
LIN {X 0,Y 440.329,Z 420.373,A -85,B 0,C 180,E1 -8950.613,E2 -8950.613} C_VEL
LIN {X 0,Y 441.262,Z 410.05,A -85,B 0,C 180,E1 -8952.293,E2 -8952.293} C_VEL
LIN {X 0,Y 442.226,Z 399.385,A -85,B 0,C 180,E1 -8953.734,E2 -8953.734} C_VEL
LIN {X 0,Y 443.15,Z 388.239,A -85,B 0,C 180,E1 -8955.001,E2 -8955.001} C_VEL
LIN {X 0,Y 444.178,Z 376.105,A -85,B 0,C 180,E1 -8956.152,E2 -8956.152} C_VEL
LIN {X 0,Y 445.262,Z 361.859,A -85,B 0,C 180,E1 -8957.257,E2 -8957.257} C_VEL
LIN {X 0,Y 446.17,Z 348.468,A -85,B 0,C 180,E1 -8958.089,E2 -8958.089} C_VEL
LIN {X 0,Y 447.012,Z 333.968,A -85,B 0,C 180,E1 -8958.793,E2 -8958.793} C_VEL
LIN {X 0,Y 447.587,Z 319.37,A -85,B 0,C 180,E1 -8959.32,E2 -8959.32} C_VEL
LIN {X 0,Y 448.07,Z 303.147,A -85,B 0,C 180,E1 -8959.702,E2 -8959.702} C_VEL
LIN {X 0,Y 450.217,Z 162.749,A -85,B 0,C 180,E1 -8962.032,E2 -8962.032} C_VEL
LIN {X 0,Y 446.238,Z 141.354,A -85,B 0,C 180,E1 -8962.673,E2 -8962.673} C_VEL
LIN {X 0,Y 442.096,Z 125.27,A -85,B 0,C 180,E1 -8964.811,E2 -8964.811} C_VEL
LIN {X 0,Y 439.439,Z 116.374,A -85,B 0,C 180,E1 -8966.042,E2 -8966.042} C_VEL
LIN {X 0,Y 439.383,Z 116.38,A -85,B 0,C 180,E1 -8969.739,E2 -8969.739} C_VEL
LIN {X 0,Y 439.444,Z 116.372,A -85,B 0,C 180,E1 -8972.367,E2 -8972.367} C_VEL
LIN {X 0,Y 439.473,Z 116.368,A -85,B 0,C 180,E1 -8974.404,E2 -8974.404} C_VEL
LIN {X 0,Y 440.444,Z 119.206,A -85,B 0,C 180,E1 -8974.525,E2 -8974.525} C_VEL
LIN {X 0,Y 449.168,Z 140.515,A -85,B 0,C 180,E1 -8975.431,E2 -8975.431} C_VEL
LIN {X 0,Y 446.608,Z 260.052,A -85,B 0,C 180,E1 -8977.719,E2 -8977.719} C_VEL
LIN {X 0,Y 446.108,Z 284.682,A -85,B 0,C 180,E1 -8978.218,E2 -8978.218} C_VEL
LIN {X 0,Y 445.612,Z 299.958,A -85,B 0,C 180,E1 -8978.704,E2 -8978.704} C_VEL
LIN {X 0,Y 444.992,Z 314.947,A -85,B 0,C 180,E1 -8979.366,E2 -8979.366} C_VEL
LIN {X 0,Y 444.287,Z 328.252,A -85,B 0,C 180,E1 -8980.117,E2 -8980.117} C_VEL
LIN {X 0,Y 443.523,Z 341.539,A -85,B 0,C 180,E1 -8981.044,E2 -8981.044} C_VEL
LIN {X 0,Y 442.718,Z 354.762,A -85,B 0,C 180,E1 -8982.171,E2 -8982.171} C_VEL
LIN {X 0,Y 441.827,Z 367.471,A -85,B 0,C 180,E1 -8983.481,E2 -8983.481} C_VEL
LIN {X 0,Y 441.127,Z 377.906,A -85,B 0,C 180,E1 -8984.759,E2 -8984.759} C_VEL
LIN {X 0,Y 440.458,Z 387.523,A -85,B 0,C 180,E1 -8986.152,E2 -8986.152} C_VEL
LIN {X 0,Y 439.913,Z 395.679,A -85,B 0,C 180,E1 -8987.545,E2 -8987.545} C_VEL
LIN {X 0,Y 439.392,Z 403.705,A -85,B 0,C 180,E1 -8989.167,E2 -8989.167} C_VEL
LIN {X 0,Y 439.043,Z 410.339,A -85,B 0,C 180,E1 -8990.788,E2 -8990.788} C_VEL
LIN {X 0,Y 438.748,Z 416.407,A -85,B 0,C 180,E1 -8992.637,E2 -8992.637} C_VEL
LIN {X 0,Y 438.589,Z 421.032,A -85,B 0,C 180,E1 -8994.482,E2 -8994.482} C_VEL
LIN {X 0,Y 438.554,Z 424.337,A -85,B 0,C 180,E1 -8996.324,E2 -8996.324} C_VEL
LIN {X 0,Y 438.405,Z 426.4,A -85,B 0,C 180,E1 -8998.162,E2 -8998.162} C_VEL
LIN {X 0,Y 438.35,Z 427.217,A -85,B 0,C 180,E1 -9000,E2 -9000} C_VEL
LIN {X 0,Y 438.467,Z 426.823,A -85,B 0,C 180,E1 -9001.837,E2 -9001.837} C_VEL
LIN {X 0,Y 438.582,Z 425.232,A -85,B 0,C 180,E1 -9003.675,E2 -9003.675} C_VEL
LIN {X 0,Y 438.597,Z 422.417,A -85,B 0,C 180,E1 -9005.517,E2 -9005.517} C_VEL
LIN {X 0,Y 438.857,Z 419.598,A -85,B 0,C 180,E1 -9006.836,E2 -9006.836} C_VEL
LIN {X 0,Y 439.155,Z 414.297,A -85,B 0,C 180,E1 -9008.744,E2 -9008.744} C_VEL
LIN {X 0,Y 439.554,Z 407.637,A -85,B 0,C 180,E1 -9010.595,E2 -9010.595} C_VEL
LIN {X 0,Y 440.121,Z 400.386,A -85,B 0,C 180,E1 -9012.215,E2 -9012.215} C_VEL
LIN {X 0,Y 440.759,Z 391.638,A -85,B 0,C 180,E1 -9013.838,E2 -9013.838} C_VEL
LIN {X 0,Y 441.535,Z 382.677,A -85,B 0,C 180,E1 -9015.226,E2 -9015.226} C_VEL
LIN {X 0,Y 442.369,Z 372.107,A -85,B 0,C 180,E1 -9016.617,E2 -9016.617} C_VEL
LIN {X 0,Y 443.351,Z 360.265,A -85,B 0,C 180,E1 -9017.915,E2 -9017.915} C_VEL
LIN {X 0,Y 444.205,Z 348.011,A -85,B 0,C 180,E1 -9019.045,E2 -9019.045} C_VEL
LIN {X 0,Y 445.173,Z 334.276,A -85,B 0,C 180,E1 -9020.082,E2 -9020.082} C_VEL
LIN {X 0,Y 446.002,Z 320.112,A -85,B 0,C 180,E1 -9020.947,E2 -9020.947} C_VEL
LIN {X 0,Y 446.769,Z 304.938,A -85,B 0,C 180,E1 -9021.666,E2 -9021.666} C_VEL
LIN {X 0,Y 447.343,Z 289.318,A -85,B 0,C 180,E1 -9022.212,E2 -9022.212} C_VEL
LIN {X 0,Y 448.054,Z 264.203,A -85,B 0,C 180,E1 -9022.783,E2 -9022.783} C_VEL
LIN {X 0,Y 450.849,Z 186.861,A -85,B 0,C 180,E1 -9024.478,E2 -9024.478} C_VEL
LIN {X 0,Y 452.608,Z 145.486,A -85,B 0,C 180,E1 -9025.446,E2 -9025.446} C_VEL
LIN {X 0,Y 447.214,Z 134.426,A -85,B 0,C 180,E1 -9026.246,E2 -9026.246} C_VEL
LIN {X 0,Y 441.907,Z 124.881,A -85,B 0,C 180,E1 -9027.082,E2 -9027.082} C_VEL
LIN {X 0,Y 439.373,Z 116.383,A -85,B 0,C 180,E1 -9029.726,E2 -9029.726} C_VEL
LIN {X 0,Y 439.37,Z 116.382,A -85,B 0,C 180,E1 -9032.946,E2 -9032.946} C_VEL
LIN {X 0,Y 439.371,Z 116.381,A -85,B 0,C 180,E1 -9036.287,E2 -9036.287} C_VEL
LIN {X 0,Y 439.357,Z 116.384,A -85,B 0,C 180,E1 -9039.78,E2 -9039.78} C_VEL
LIN {X 0,Y 439.332,Z 116.385,A -85,B 0,C 180,E1 -9042.62,E2 -9042.62} C_VEL
LIN {X 0,Y 439.396,Z 116.379,A -85,B 0,C 180,E1 -9045.27,E2 -9045.27} C_VEL
LIN {X 0,Y 439.352,Z 116.385,A -85,B 0,C 180,E1 -9049.016,E2 -9049.016} C_VEL
LIN {X 0,Y 439.343,Z 116.388,A -85,B 0,C 180,E1 -9052.564,E2 -9052.564} C_VEL
LIN {X 0,Y 439.393,Z 116.465,A -85,B 0,C 180,E1 -9054.584,E2 -9054.584} C_VEL
LIN {X 0,Y 442.386,Z 125.658,A -85,B 0,C 180,E1 -9057.036,E2 -9057.036} C_VEL
LIN {X 0,Y 444.957,Z 135.298,A -85,B 0,C 180,E1 -9059.219,E2 -9059.219} C_VEL
LIN {X 0,Y 446.6,Z 143.143,A -85,B 0,C 180,E1 -9060.801,E2 -9060.801} C_VEL
LIN {X 0,Y 445.122,Z 158.215,A -85,B 0,C 180,E1 -9063.238,E2 -9063.238} C_VEL
LIN {X 0,Y 449.087,Z 178.14,A -85,B 0,C 180,E1 -9064.156,E2 -9064.156} C_VEL
LIN {X 0,Y 451.339,Z 194.858,A -85,B 0,C 180,E1 -9064.789,E2 -9064.789} C_VEL
LIN {X 0,Y 448.175,Z 281.392,A -85,B 0,C 180,E1 -9066.705,E2 -9066.705} C_VEL
LIN {X 0,Y 446.833,Z 329.496,A -85,B 0,C 180,E1 -9067.731,E2 -9067.731} C_VEL
LIN {X 0,Y 445.928,Z 346.14,A -85,B 0,C 180,E1 -9068.262,E2 -9068.262} C_VEL
LIN {X 0,Y 445.23,Z 362.255,A -85,B 0,C 180,E1 -9068.894,E2 -9068.894} C_VEL
LIN {X 0,Y 444.374,Z 376.522,A -85,B 0,C 180,E1 -9069.639,E2 -9069.639} C_VEL
LIN {X 0,Y 443.597,Z 388.766,A -85,B 0,C 180,E1 -9070.446,E2 -9070.446} C_VEL
LIN {X 0,Y 442.656,Z 401.693,A -85,B 0,C 180,E1 -9071.486,E2 -9071.486} C_VEL
LIN {X 0,Y 441.769,Z 413.676,A -85,B 0,C 180,E1 -9072.654,E2 -9072.654} C_VEL
LIN {X 0,Y 440.88,Z 425.473,A -85,B 0,C 180,E1 -9074.039,E2 -9074.039} C_VEL
LIN {X 0,Y 440.129,Z 435.435,A -85,B 0,C 180,E1 -9075.434,E2 -9075.434} C_VEL
LIN {X 0,Y 439.461,Z 445.144,A -85,B 0,C 180,E1 -9077.062,E2 -9077.062} C_VEL
LIN {X 0,Y 439.022,Z 453.201,A -85,B 0,C 180,E1 -9078.691,E2 -9078.691} C_VEL
LIN {X 0,Y 438.641,Z 459.871,A -85,B 0,C 180,E1 -9080.315,E2 -9080.315} C_VEL
LIN {X 0,Y 438.468,Z 465.973,A -85,B 0,C 180,E1 -9082.17,E2 -9082.17} C_VEL
LIN {X 0,Y 438.42,Z 469.788,A -85,B 0,C 180,E1 -9083.655,E2 -9083.655} C_VEL
LIN {X 0,Y 438.323,Z 473.217,A -85,B 0,C 180,E1 -9085.402,E2 -9085.402} C_VEL
LIN {X 0,Y 438.37,Z 475.626,A -85,B 0,C 180,E1 -9087.243,E2 -9087.243} C_VEL
LIN {X 0,Y 438.258,Z 476.831,A -85,B 0,C 180,E1 -9089.081,E2 -9089.081} C_VEL
LIN {X 0,Y 438.257,Z 476.837,A -85,B 0,C 180,E1 -9090.919,E2 -9090.919} C_VEL
LIN {X 0,Y 438.366,Z 475.63,A -85,B 0,C 180,E1 -9092.757,E2 -9092.757} C_VEL
LIN {X 0,Y 438.321,Z 473.213,A -85,B 0,C 180,E1 -9094.598,E2 -9094.598} C_VEL
LIN {X 0,Y 438.428,Z 469.537,A -85,B 0,C 180,E1 -9096.443,E2 -9096.443} C_VEL
LIN {X 0,Y 438.513,Z 464.51,A -85,B 0,C 180,E1 -9098.293,E2 -9098.293} C_VEL
LIN {X 0,Y 438.701,Z 458.001,A -85,B 0,C 180,E1 -9100.15,E2 -9100.15} C_VEL
LIN {X 0,Y 439.076,Z 450.937,A -85,B 0,C 180,E1 -9101.776,E2 -9101.776} C_VEL
LIN {X 0,Y 439.57,Z 442.385,A -85,B 0,C 180,E1 -9103.405,E2 -9103.405} C_VEL
LIN {X 0,Y 440.305,Z 432.038,A -85,B 0,C 180,E1 -9105.033,E2 -9105.033} C_VEL
LIN {X 0,Y 441.119,Z 421.387,A -85,B 0,C 180,E1 -9106.427,E2 -9106.427} C_VEL
LIN {X 0,Y 441.873,Z 410.9,A -85,B 0,C 180,E1 -9107.59,E2 -9107.59} C_VEL
LIN {X 0,Y 442.757,Z 398.376,A -85,B 0,C 180,E1 -9108.75,E2 -9108.75} C_VEL
LIN {X 0,Y 443.707,Z 384.575,A -85,B 0,C 180,E1 -9109.789,E2 -9109.789} C_VEL
LIN {X 0,Y 444.609,Z 370.343,A -85,B 0,C 180,E1 -9110.639,E2 -9110.639} C_VEL
LIN {X 0,Y 445.313,Z 355.584,A -85,B 0,C 180,E1 -9111.317,E2 -9111.317} C_VEL
LIN {X 0,Y 445.856,Z 340.916,A -85,B 0,C 180,E1 -9111.802,E2 -9111.802} C_VEL
LIN {X 0,Y 446.187,Z 324.44,A -85,B 0,C 180,E1 -9112.151,E2 -9112.151} C_VEL
LIN {X 0,Y 448.319,Z 252.489,A -85,B 0,C 180,E1 -9113.654,E2 -9113.654} C_VEL
LIN {X 0,Y 450.483,Z 189.371,A -85,B 0,C 180,E1 -9115.101,E2 -9115.101} C_VEL
LIN {X 0,Y 447.451,Z 163.893,A -85,B 0,C 180,E1 -9116.048,E2 -9116.048} C_VEL
LIN {X 0,Y 445.844,Z 152.809,A -85,B 0,C 180,E1 -9116.532,E2 -9116.532} C_VEL
LIN {X 0,Y 446.515,Z 143.597,A -85,B 0,C 180,E1 -9117.57,E2 -9117.57} C_VEL
LIN {X 0,Y 445.867,Z 139.969,A -85,B 0,C 180,E1 -9118.03,E2 -9118.03} C_VEL
LIN {X 0,Y 439.816,Z 118.036,A -85,B 0,C 180,E1 -9121.02,E2 -9121.02} C_VEL
LIN {X 0,Y 439.396,Z 116.379,A -85,B 0,C 180,E1 -9121.254,E2 -9121.254} C_VEL
LIN {X 0,Y 439.357,Z 116.38,A -85,B 0,C 180,E1 -9124.046,E2 -9124.046} C_VEL
LIN {X 0,Y 439.345,Z 116.384,A -85,B 0,C 180,E1 -9126.887,E2 -9126.887} C_VEL
LIN {X 0,Y 439.346,Z 116.383,A -85,B 0,C 180,E1 -9129.841,E2 -9129.841} C_VEL
LIN {X 0,Y 439.331,Z 116.384,A -85,B 0,C 180,E1 -9132.62,E2 -9132.62} C_VEL
LIN {X 0,Y 439.396,Z 116.373,A -85,B 0,C 180,E1 -9135.27,E2 -9135.27} C_VEL
LIN {X 0,Y 439.352,Z 116.381,A -85,B 0,C 180,E1 -9139.016,E2 -9139.016} C_VEL
LIN {X 0,Y 439.344,Z 116.384,A -85,B 0,C 180,E1 -9142.565,E2 -9142.565} C_VEL
LIN {X 0,Y 439.394,Z 116.38,A -85,B 0,C 180,E1 -9144.844,E2 -9144.844} C_VEL
LIN {X 0,Y 439.369,Z 116.382,A -85,B 0,C 180,E1 -9148.139,E2 -9148.139} C_VEL
LIN {X 0,Y 439.4,Z 116.379,A -85,B 0,C 180,E1 -9151.606,E2 -9151.606} C_VEL
LIN {X 0,Y 439.439,Z 116.546,A -85,B 0,C 180,E1 -9151.961,E2 -9151.961} C_VEL
LIN {X 0,Y 441.397,Z 121.91,A -85,B 0,C 180,E1 -9152.974,E2 -9152.974} C_VEL
LIN {X 0,Y 447.707,Z 133.569,A -85,B 0,C 180,E1 -9153.95,E2 -9153.95} C_VEL
LIN {X 0,Y 452.492,Z 144.359,A -85,B 0,C 180,E1 -9154.676,E2 -9154.676} C_VEL
LIN {X 0,Y 448.948,Z 232.088,A -85,B 0,C 180,E1 -9156.656,E2 -9156.656} C_VEL
LIN {X 0,Y 447.329,Z 287.21,A -85,B 0,C 180,E1 -9157.848,E2 -9157.848} C_VEL
LIN {X 0,Y 446.749,Z 302.888,A -85,B 0,C 180,E1 -9158.368,E2 -9158.368} C_VEL
LIN {X 0,Y 446.018,Z 317.905,A -85,B 0,C 180,E1 -9159.054,E2 -9159.054} C_VEL
LIN {X 0,Y 445.309,Z 330.671,A -85,B 0,C 180,E1 -9159.804,E2 -9159.804} C_VEL
LIN {X 0,Y 444.374,Z 345.097,A -85,B 0,C 180,E1 -9160.842,E2 -9160.842} C_VEL
LIN {X 0,Y 443.394,Z 358.109,A -85,B 0,C 180,E1 -9161.995,E2 -9161.995} C_VEL
LIN {X 0,Y 442.482,Z 369.047,A -85,B 0,C 180,E1 -9163.15,E2 -9163.15} C_VEL
LIN {X 0,Y 441.705,Z 380.085,A -85,B 0,C 180,E1 -9164.544,E2 -9164.544} C_VEL
LIN {X 0,Y 440.817,Z 390.831,A -85,B 0,C 180,E1 -9166.164,E2 -9166.164} C_VEL
LIN {X 0,Y 440.109,Z 399.693,A -85,B 0,C 180,E1 -9167.785,E2 -9167.785} C_VEL
LIN {X 0,Y 439.589,Z 407.022,A -85,B 0,C 180,E1 -9169.406,E2 -9169.406} C_VEL
LIN {X 0,Y 439.149,Z 413.794,A -85,B 0,C 180,E1 -9171.255,E2 -9171.255} C_VEL
LIN {X 0,Y 438.878,Z 417.823,A -85,B 0,C 180,E1 -9172.64,E2 -9172.64} C_VEL
LIN {X 0,Y 438.813,Z 420.087,A -85,B 0,C 180,E1 -9173.563,E2 -9173.563} C_VEL
LIN {X 0,Y 438.53,Z 423.633,A -85,B 0,C 180,E1 -9175.404,E2 -9175.404} C_VEL
LIN {X 0,Y 438.513,Z 425.903,A -85,B 0,C 180,E1 -9177.244,E2 -9177.244} C_VEL
LIN {X 0,Y 438.374,Z 426.967,A -85,B 0,C 180,E1 -9179.082,E2 -9179.082} C_VEL
LIN {X 0,Y 438.373,Z 426.817,A -85,B 0,C 180,E1 -9180.919,E2 -9180.919} C_VEL
LIN {X 0,Y 438.469,Z 425.432,A -85,B 0,C 180,E1 -9182.756,E2 -9182.756} C_VEL
LIN {X 0,Y 438.448,Z 422.821,A -85,B 0,C 180,E1 -9184.597,E2 -9184.597} C_VEL
LIN {X 0,Y 438.681,Z 418.923,A -85,B 0,C 180,E1 -9186.439,E2 -9186.439} C_VEL
LIN {X 0,Y 438.879,Z 413.662,A -85,B 0,C 180,E1 -9188.287,E2 -9188.287} C_VEL
LIN {X 0,Y 439.202,Z 406.894,A -85,B 0,C 180,E1 -9190.138,E2 -9190.138} C_VEL
LIN {X 0,Y 439.754,Z 398.412,A -85,B 0,C 180,E1 -9191.992,E2 -9191.992} C_VEL
LIN {X 0,Y 440.264,Z 389.313,A -85,B 0,C 180,E1 -9193.619,E2 -9193.619} C_VEL
LIN {X 0,Y 441.04,Z 378.308,A -85,B 0,C 180,E1 -9195.244,E2 -9195.244} C_VEL
LIN {X 0,Y 441.833,Z 366.962,A -85,B 0,C 180,E1 -9196.638,E2 -9196.638} C_VEL
LIN {X 0,Y 442.673,Z 354.509,A -85,B 0,C 180,E1 -9197.915,E2 -9197.915} C_VEL
LIN {X 0,Y 443.526,Z 340.789,A -85,B 0,C 180,E1 -9199.076,E2 -9199.076} C_VEL
LIN {X 0,Y 444.309,Z 327.393,A -85,B 0,C 180,E1 -9200.003,E2 -9200.003} C_VEL
LIN {X 0,Y 445.1,Z 312.735,A -85,B 0,C 180,E1 -9200.81,E2 -9200.81} C_VEL
LIN {X 0,Y 445.669,Z 297.744,A -85,B 0,C 180,E1 -9201.446,E2 -9201.446} C_VEL
LIN {X 0,Y 446.117,Z 281.859,A -85,B 0,C 180,E1 -9201.924,E2 -9201.924} C_VEL
LIN {X 0,Y 449.099,Z 141.308,A -85,B 0,C 180,E1 -9204.615,E2 -9204.615} C_VEL
LIN {X 0,Y 440.245,Z 118.891,A -85,B 0,C 180,E1 -9205.553,E2 -9205.553} C_VEL
LIN {X 0,Y 439.445,Z 116.373,A -85,B 0,C 180,E1 -9205.673,E2 -9205.673} C_VEL
LIN {X 0,Y 439.392,Z 116.376,A -85,B 0,C 180,E1 -9208.676,E2 -9208.676} C_VEL
LIN {X 0,Y 439.368,Z 116.381,A -85,B 0,C 180,E1 -9212.03,E2 -9212.03} C_VEL
LIN {X 0,Y 439.393,Z 116.379,A -85,B 0,C 180,E1 -9215.34,E2 -9215.34} C_VEL
LIN {X 0,Y 439.364,Z 116.378,A -85,B 0,C 180,E1 -9218.597,E2 -9218.597} C_VEL
LIN {X 0,Y 439.353,Z 116.379,A -85,B 0,C 180,E1 -9222.21,E2 -9222.21} C_VEL
LIN {X 0,Y 439.399,Z 116.365,A -85,B 0,C 180,E1 -9225.27,E2 -9225.27} C_VEL
LIN {X 0,Y 439.355,Z 116.377,A -85,B 0,C 180,E1 -9229.016,E2 -9229.016} C_VEL
LIN {X 0,Y 439.369,Z 116.377,A -85,B 0,C 180,E1 -9231.609,E2 -9231.609} C_VEL
LIN {X 0,Y 439.397,Z 116.363,A -85,B 0,C 180,E1 -9234.844,E2 -9234.844} C_VEL
LIN {X 0,Y 439.368,Z 116.378,A -85,B 0,C 180,E1 -9238.139,E2 -9238.139} C_VEL
LIN {X 0,Y 439.403,Z 116.371,A -85,B 0,C 180,E1 -9241.606,E2 -9241.606} C_VEL
LIN {X 0,Y 439.369,Z 116.381,A -85,B 0,C 180,E1 -9244.413,E2 -9244.413} C_VEL
LIN {X 0,Y 439.363,Z 116.379,A -85,B 0,C 180,E1 -9247.424,E2 -9247.424} C_VEL
LIN {X 0,Y 439.377,Z 116.372,A -85,B 0,C 180,E1 -9249.647,E2 -9249.647} C_VEL
LIN {X 0,Y 438.706,Z 116.458,A -85,B 0,C 180,E1 -9250.412,E2 -9250.412} C_VEL
LIN {X 0,Y 435.843,Z 116.817,A -85,B 0,C 180,E1 -9251.655,E2 -9251.655} C_VEL
LIN {X 0,Y 433.442,Z 117.119,A -85,B 0,C 180,E1 -9252.658,E2 -9252.658} C_VEL
LIN {X 0,Y 432.438,Z 117.238,A -85,B 0,C 180,E1 -9253.433,E2 -9253.433} C_VEL
LIN {X 0,Y 432.371,Z 117.245,A -85,B 0,C 180,E1 -9253.695,E2 -9253.695} C_VEL
LIN {X 0,Y 432.434,Z 117.242,A -85,B 0,C 180,E1 -9257.197,E2 -9257.197} C_VEL
LIN {X 0,Y 432.428,Z 117.247,A -85,B 0,C 180,E1 -9260.647,E2 -9260.647} C_VEL
LIN {X 0,Y 432.514,Z 117.234,A -85,B 0,C 180,E1 -9263.469,E2 -9263.469} C_VEL
LIN {X 0,Y 432.375,Z 117.252,A -85,B 0,C 180,E1 -9265.338,E2 -9265.338} C_VEL
LIN {X 0,Y 432.467,Z 117.244,A -85,B 0,C 180,E1 -9266.914,E2 -9266.914} C_VEL
LIN {X 0,Y 435.792,Z 130.347,A -85,B 0,C 180,E1 -9269.109,E2 -9269.109} C_VEL
LIN {X 0,Y 437.836,Z 140.209,A -85,B 0,C 180,E1 -9270.714,E2 -9270.714} C_VEL
LIN {X 0,Y 437.817,Z 142.792,A -85,B 0,C 180,E1 -9271.092,E2 -9271.092} C_VEL
LIN {X 0,Y 443.302,Z 168.294,A -85,B 0,C 180,E1 -9271.881,E2 -9271.881} C_VEL
LIN {X 0,Y 441.043,Z 309.255,A -85,B 0,C 180,E1 -9274.255,E2 -9274.255} C_VEL
LIN {X 0,Y 440.538,Z 324.531,A -85,B 0,C 180,E1 -9274.69,E2 -9274.69} C_VEL
LIN {X 0,Y 439.869,Z 338.817,A -85,B 0,C 180,E1 -9275.271,E2 -9275.271} C_VEL
LIN {X 0,Y 439.023,Z 352.692,A -85,B 0,C 180,E1 -9276.012,E2 -9276.012} C_VEL
LIN {X 0,Y 438.09,Z 366.024,A -85,B 0,C 180,E1 -9276.91,E2 -9276.91} C_VEL
LIN {X 0,Y 437.039,Z 378.876,A -85,B 0,C 180,E1 -9277.973,E2 -9277.973} C_VEL
LIN {X 0,Y 435.928,Z 391.807,A -85,B 0,C 180,E1 -9279.278,E2 -9279.278} C_VEL
LIN {X 0,Y 435.052,Z 401.748,A -85,B 0,C 180,E1 -9280.471,E2 -9280.471} C_VEL
LIN {X 0,Y 434.098,Z 411.927,A -85,B 0,C 180,E1 -9281.913,E2 -9281.913} C_VEL
LIN {X 0,Y 433.215,Z 422.051,A -85,B 0,C 180,E1 -9283.633,E2 -9283.633} C_VEL
LIN {X 0,Y 432.533,Z 430.18,A -85,B 0,C 180,E1 -9285.31,E2 -9285.31} C_VEL
LIN {X 0,Y 432.036,Z 437.017,A -85,B 0,C 180,E1 -9287.026,E2 -9287.026} C_VEL
LIN {X 0,Y 431.624,Z 443.332,A -85,B 0,C 180,E1 -9289.005,E2 -9289.005} C_VEL
LIN {X 0,Y 431.343,Z 448.157,A -85,B 0,C 180,E1 -9291.005,E2 -9291.005} C_VEL
LIN {X 0,Y 431.113,Z 451.579,A -85,B 0,C 180,E1 -9293.032,E2 -9293.032} C_VEL
LIN {X 0,Y 431.016,Z 453.616,A -85,B 0,C 180,E1 -9295.084,E2 -9295.084} C_VEL
LIN {X 0,Y 431.013,Z 454.267,A -85,B 0,C 180,E1 -9297.166,E2 -9297.166} C_VEL
LIN {X 0,Y 431.026,Z 454.018,A -85,B 0,C 180,E1 -9298.298,E2 -9298.298} C_VEL
LIN {X 0,Y 431.122,Z 452.516,A -85,B 0,C 180,E1 -9300.355,E2 -9300.355} C_VEL
LIN {X 0,Y 431.239,Z 450.223,A -85,B 0,C 180,E1 -9302.063,E2 -9302.063} C_VEL
LIN {X 0,Y 431.463,Z 446.755,A -85,B 0,C 180,E1 -9303.826,E2 -9303.826} C_VEL
LIN {X 0,Y 431.7,Z 442.39,A -85,B 0,C 180,E1 -9305.512,E2 -9305.512} C_VEL
LIN {X 0,Y 432.052,Z 437.096,A -85,B 0,C 180,E1 -9307.149,E2 -9307.149} C_VEL
LIN {X 0,Y 432.655,Z 429.736,A -85,B 0,C 180,E1 -9308.985,E2 -9308.985} C_VEL
LIN {X 0,Y 433.345,Z 421.054,A -85,B 0,C 180,E1 -9310.751,E2 -9310.751} C_VEL
LIN {X 0,Y 434.223,Z 412.082,A -85,B 0,C 180,E1 -9312.268,E2 -9312.268} C_VEL
LIN {X 0,Y 435.218,Z 401.491,A -85,B 0,C 180,E1 -9313.768,E2 -9313.768} C_VEL
LIN {X 0,Y 436.246,Z 389.899,A -85,B 0,C 180,E1 -9315.141,E2 -9315.141} C_VEL
LIN {X 0,Y 437.315,Z 377.969,A -85,B 0,C 180,E1 -9316.318,E2 -9316.318} C_VEL
LIN {X 0,Y 438.45,Z 364.343,A -85,B 0,C 180,E1 -9317.421,E2 -9317.421} C_VEL
LIN {X 0,Y 439.473,Z 350.134,A -85,B 0,C 180,E1 -9318.344,E2 -9318.344} C_VEL
LIN {X 0,Y 440.315,Z 337.064,A -85,B 0,C 180,E1 -9319.015,E2 -9319.015} C_VEL
LIN {X 0,Y 440.95,Z 321.96,A -85,B 0,C 180,E1 -9319.602,E2 -9319.602} C_VEL
LIN {X 0,Y 441.475,Z 306.802,A -85,B 0,C 180,E1 -9319.996,E2 -9319.996} C_VEL
LIN {X 0,Y 443.855,Z 163.863,A -85,B 0,C 180,E1 -9322.409,E2 -9322.409} C_VEL
LIN {X 0,Y 440.078,Z 143.868,A -85,B 0,C 180,E1 -9323.018,E2 -9323.018} C_VEL
LIN {X 0,Y 439.156,Z 141.329,A -85,B 0,C 180,E1 -9323.147,E2 -9323.147} C_VEL
LIN {X 0,Y 435.458,Z 127.338,A -85,B 0,C 180,E1 -9325.044,E2 -9325.044} C_VEL
LIN {X 0,Y 432.365,Z 117.252,A -85,B 0,C 180,E1 -9326.485,E2 -9326.485} C_VEL
LIN {X 0,Y 432.348,Z 117.256,A -85,B 0,C 180,E1 -9329.74,E2 -9329.74} C_VEL
LIN {X 0,Y 432.394,Z 117.251,A -85,B 0,C 180,E1 -9332.928,E2 -9332.928} C_VEL
LIN {X 0,Y 432.443,Z 117.244,A -85,B 0,C 180,E1 -9334.022,E2 -9334.022} C_VEL
LIN {X 0,Y 434.073,Z 121.721,A -85,B 0,C 180,E1 -9334.23,E2 -9334.23} C_VEL
LIN {X 0,Y 441.511,Z 139.714,A -85,B 0,C 180,E1 -9335.018,E2 -9335.018} C_VEL
LIN {X 0,Y 442.645,Z 142.963,A -85,B 0,C 180,E1 -9335.146,E2 -9335.146} C_VEL
LIN {X 0,Y 439.37,Z 283.63,A -85,B 0,C 180,E1 -9337.913,E2 -9337.913} C_VEL
LIN {X 0,Y 438.857,Z 299.565,A -85,B 0,C 180,E1 -9338.418,E2 -9338.418} C_VEL
LIN {X 0,Y 438.202,Z 314.783,A -85,B 0,C 180,E1 -9339.093,E2 -9339.093} C_VEL
LIN {X 0,Y 437.417,Z 329.074,A -85,B 0,C 180,E1 -9339.913,E2 -9339.913} C_VEL
LIN {X 0,Y 436.625,Z 342.279,A -85,B 0,C 180,E1 -9340.855,E2 -9340.855} C_VEL
LIN {X 0,Y 435.85,Z 354.61,A -85,B 0,C 180,E1 -9341.917,E2 -9341.917} C_VEL
LIN {X 0,Y 434.954,Z 367.125,A -85,B 0,C 180,E1 -9343.212,E2 -9343.212} C_VEL
LIN {X 0,Y 434.073,Z 379.371,A -85,B 0,C 180,E1 -9344.746,E2 -9344.746} C_VEL
LIN {X 0,Y 433.397,Z 388.884,A -85,B 0,C 180,E1 -9346.161,E2 -9346.161} C_VEL
LIN {X 0,Y 432.813,Z 398.161,A -85,B 0,C 180,E1 -9347.813,E2 -9347.813} C_VEL
LIN {X 0,Y 432.217,Z 406.813,A -85,B 0,C 180,E1 -9349.696,E2 -9349.696} C_VEL
LIN {X 0,Y 431.855,Z 413.738,A -85,B 0,C 180,E1 -9351.578,E2 -9351.578} C_VEL
LIN {X 0,Y 431.568,Z 419.136,A -85,B 0,C 180,E1 -9353.454,E2 -9353.454} C_VEL
LIN {X 0,Y 431.39,Z 423.15,A -85,B 0,C 180,E1 -9355.327,E2 -9355.327} C_VEL
LIN {X 0,Y 431.411,Z 425.872,A -85,B 0,C 180,E1 -9357.198,E2 -9357.198} C_VEL
LIN {X 0,Y 431.285,Z 427.344,A -85,B 0,C 180,E1 -9359.066,E2 -9359.066} C_VEL
LIN {X 0,Y 431.317,Z 427.596,A -85,B 0,C 180,E1 -9360.933,E2 -9360.933} C_VEL
LIN {X 0,Y 431.444,Z 426.64,A -85,B 0,C 180,E1 -9362.801,E2 -9362.801} C_VEL
LIN {X 0,Y 431.49,Z 424.479,A -85,B 0,C 180,E1 -9364.671,E2 -9364.671} C_VEL
LIN {X 0,Y 431.783,Z 421.04,A -85,B 0,C 180,E1 -9366.542,E2 -9366.542} C_VEL
LIN {X 0,Y 432.027,Z 416.264,A -85,B 0,C 180,E1 -9368.419,E2 -9368.419} C_VEL
LIN {X 0,Y 432.473,Z 410.027,A -85,B 0,C 180,E1 -9370.297,E2 -9370.297} C_VEL
LIN {X 0,Y 433.084,Z 402.117,A -85,B 0,C 180,E1 -9372.178,E2 -9372.178} C_VEL
LIN {X 0,Y 433.793,Z 393.556,A -85,B 0,C 180,E1 -9373.841,E2 -9373.841} C_VEL
LIN {X 0,Y 434.712,Z 383.377,A -85,B 0,C 180,E1 -9375.471,E2 -9375.471} C_VEL
LIN {X 0,Y 435.599,Z 372.859,A -85,B 0,C 180,E1 -9376.882,E2 -9376.882} C_VEL
LIN {X 0,Y 436.657,Z 361.234,A -85,B 0,C 180,E1 -9378.184,E2 -9378.184} C_VEL
LIN {X 0,Y 437.566,Z 348.934,A -85,B 0,C 180,E1 -9379.346,E2 -9379.346} C_VEL
LIN {X 0,Y 438.609,Z 335.346,A -85,B 0,C 180,E1 -9380.396,E2 -9380.396} C_VEL
LIN {X 0,Y 439.462,Z 321.4,A -85,B 0,C 180,E1 -9381.274,E2 -9381.274} C_VEL
LIN {X 0,Y 440.336,Z 306.054,A -85,B 0,C 180,E1 -9382.022,E2 -9382.022} C_VEL
LIN {X 0,Y 440.968,Z 290.614,A -85,B 0,C 180,E1 -9382.581,E2 -9382.581} C_VEL
LIN {X 0,Y 441.64,Z 267.688,A -85,B 0,C 180,E1 -9383.132,E2 -9383.132} C_VEL
LIN {X 0,Y 444.584,Z 191.797,A -85,B 0,C 180,E1 -9384.851,E2 -9384.851} C_VEL
LIN {X 0,Y 446.621,Z 147.669,A -85,B 0,C 180,E1 -9385.914,E2 -9385.914} C_VEL
LIN {X 0,Y 440.627,Z 135.658,A -85,B 0,C 180,E1 -9386.861,E2 -9386.861} C_VEL
LIN {X 0,Y 436.292,Z 128.387,A -85,B 0,C 180,E1 -9387.554,E2 -9387.554} C_VEL
LIN {X 0,Y 434.955,Z 125.791,A -85,B 0,C 180,E1 -9387.816,E2 -9387.816} C_VEL
LIN {X 0,Y 432.334,Z 117.259,A -85,B 0,C 180,E1 -9390.707,E2 -9390.707} C_VEL
LIN {X 0,Y 432.332,Z 117.258,A -85,B 0,C 180,E1 -9393.998,E2 -9393.998} C_VEL
LIN {X 0,Y 432.319,Z 117.26,A -85,B 0,C 180,E1 -9397.196,E2 -9397.196} C_VEL
LIN {X 0,Y 432.289,Z 117.263,A -85,B 0,C 180,E1 -9400.172,E2 -9400.172} C_VEL
LIN {X 0,Y 432.301,Z 117.262,A -85,B 0,C 180,E1 -9403.063,E2 -9403.063} C_VEL
LIN {X 0,Y 432.332,Z 117.258,A -85,B 0,C 180,E1 -9405.665,E2 -9405.665} C_VEL
LIN {X 0,Y 432.306,Z 117.261,A -85,B 0,C 180,E1 -9408.402,E2 -9408.402} C_VEL
LIN {X 0,Y 432.328,Z 117.259,A -85,B 0,C 180,E1 -9411.849,E2 -9411.849} C_VEL
LIN {X 0,Y 432.357,Z 117.375,A -85,B 0,C 180,E1 -9413.644,E2 -9413.644} C_VEL
LIN {X 0,Y 435.291,Z 126.252,A -85,B 0,C 180,E1 -9416.233,E2 -9416.233} C_VEL
LIN {X 0,Y 437.705,Z 134.74,A -85,B 0,C 180,E1 -9418.32,E2 -9418.32} C_VEL
LIN {X 0,Y 439.801,Z 143.968,A -85,B 0,C 180,E1 -9420.305,E2 -9420.305} C_VEL
LIN {X 0,Y 439.946,Z 146.865,A -85,B 0,C 180,E1 -9420.841,E2 -9420.841} C_VEL
LIN {X 0,Y 438.795,Z 157.844,A -85,B 0,C 180,E1 -9422.62,E2 -9422.62} C_VEL
LIN {X 0,Y 442.754,Z 177.273,A -85,B 0,C 180,E1 -9423.584,E2 -9423.584} C_VEL
LIN {X 0,Y 445.247,Z 194.786,A -85,B 0,C 180,E1 -9424.292,E2 -9424.292} C_VEL
LIN {X 0,Y 442.414,Z 267.4,A -85,B 0,C 180,E1 -9425.979,E2 -9425.979} C_VEL
LIN {X 0,Y 440.361,Z 329.707,A -85,B 0,C 180,E1 -9427.355,E2 -9427.355} C_VEL
LIN {X 0,Y 439.399,Z 346.127,A -85,B 0,C 180,E1 -9427.903,E2 -9427.903} C_VEL
LIN {X 0,Y 438.516,Z 364.024,A -85,B 0,C 180,E1 -9428.637,E2 -9428.637} C_VEL
LIN {X 0,Y 437.578,Z 378.465,A -85,B 0,C 180,E1 -9429.431,E2 -9429.431} C_VEL
LIN {X 0,Y 436.699,Z 391.844,A -85,B 0,C 180,E1 -9430.37,E2 -9430.37} C_VEL
LIN {X 0,Y 435.582,Z 405.434,A -85,B 0,C 180,E1 -9431.54,E2 -9431.54} C_VEL
LIN {X 0,Y 434.595,Z 417.962,A -85,B 0,C 180,E1 -9432.865,E2 -9432.865} C_VEL
LIN {X 0,Y 433.685,Z 428.883,A -85,B 0,C 180,E1 -9434.25,E2 -9434.25} C_VEL
LIN {X 0,Y 432.962,Z 438.276,A -85,B 0,C 180,E1 -9435.668,E2 -9435.668} C_VEL
LIN {X 0,Y 432.299,Z 447.217,A -85,B 0,C 180,E1 -9437.273,E2 -9437.273} C_VEL
LIN {X 0,Y 431.884,Z 455.075,A -85,B 0,C 180,E1 -9438.977,E2 -9438.977} C_VEL
LIN {X 0,Y 431.526,Z 461.339,A -85,B 0,C 180,E1 -9440.627,E2 -9440.627} C_VEL
LIN {X 0,Y 431.375,Z 467.06,A -85,B 0,C 180,E1 -9442.511,E2 -9442.511} C_VEL
LIN {X 0,Y 431.255,Z 471.372,A -85,B 0,C 180,E1 -9444.389,E2 -9444.389} C_VEL
LIN {X 0,Y 431.193,Z 474.392,A -85,B 0,C 180,E1 -9446.262,E2 -9446.262} C_VEL
LIN {X 0,Y 431.262,Z 476.194,A -85,B 0,C 180,E1 -9448.132,E2 -9448.132} C_VEL
LIN {X 0,Y 431.172,Z 476.803,A -85,B 0,C 180,E1 -9450,E2 -9450} C_VEL
LIN {X 0,Y 431.26,Z 476.195,A -85,B 0,C 180,E1 -9451.868,E2 -9451.868} C_VEL
LIN {X 0,Y 431.201,Z 474.381,A -85,B 0,C 180,E1 -9453.738,E2 -9453.738} C_VEL
LIN {X 0,Y 431.269,Z 471.338,A -85,B 0,C 180,E1 -9455.611,E2 -9455.611} C_VEL
LIN {X 0,Y 431.375,Z 466.993,A -85,B 0,C 180,E1 -9457.489,E2 -9457.489} C_VEL
LIN {X 0,Y 431.513,Z 461.236,A -85,B 0,C 180,E1 -9459.373,E2 -9459.373} C_VEL
LIN {X 0,Y 431.939,Z 453.908,A -85,B 0,C 180,E1 -9461.259,E2 -9461.259} C_VEL
LIN {X 0,Y 432.299,Z 446.492,A -85,B 0,C 180,E1 -9462.822,E2 -9462.822} C_VEL
LIN {X 0,Y 432.907,Z 437.951,A -85,B 0,C 180,E1 -9464.334,E2 -9464.334} C_VEL
LIN {X 0,Y 433.638,Z 428.468,A -85,B 0,C 180,E1 -9465.752,E2 -9465.752} C_VEL
LIN {X 0,Y 434.404,Z 417.756,A -85,B 0,C 180,E1 -9467.101,E2 -9467.101} C_VEL
LIN {X 0,Y 435.435,Z 404.628,A -85,B 0,C 180,E1 -9468.467,E2 -9468.467} C_VEL
LIN {X 0,Y 436.422,Z 392.309,A -85,B 0,C 180,E1 -9469.521,E2 -9469.521} C_VEL
LIN {X 0,Y 437.331,Z 378.9,A -85,B 0,C 180,E1 -9470.458,E2 -9470.458} C_VEL
LIN {X 0,Y 438.325,Z 364.093,A -85,B 0,C 180,E1 -9471.264,E2 -9471.264} C_VEL
LIN {X 0,Y 438.904,Z 350.508,A -85,B 0,C 180,E1 -9471.832,E2 -9471.832} C_VEL
LIN {X 0,Y 439.4,Z 335.832,A -85,B 0,C 180,E1 -9472.263,E2 -9472.263} C_VEL
LIN {X 0,Y 442.599,Z 237.59,A -85,B 0,C 180,E1 -9474.444,E2 -9474.444} C_VEL
LIN {X 0,Y 444.444,Z 190.27,A -85,B 0,C 180,E1 -9475.57,E2 -9475.57} C_VEL
LIN {X 0,Y 441.595,Z 165.111,A -85,B 0,C 180,E1 -9476.547,E2 -9476.547} C_VEL
LIN {X 0,Y 439.339,Z 149.567,A -85,B 0,C 180,E1 -9477.252,E2 -9477.252} C_VEL
LIN {X 0,Y 439.602,Z 143.749,A -85,B 0,C 180,E1 -9477.928,E2 -9477.928} C_VEL
LIN {X 0,Y 433.498,Z 121.455,A -85,B 0,C 180,E1 -9480.998,E2 -9480.998} C_VEL
LIN {X 0,Y 432.349,Z 117.257,A -85,B 0,C 180,E1 -9481.617,E2 -9481.617} C_VEL
LIN {X 0,Y 432.326,Z 117.26,A -85,B 0,C 180,E1 -9484.678,E2 -9484.678} C_VEL
LIN {X 0,Y 432.328,Z 117.258,A -85,B 0,C 180,E1 -9488.151,E2 -9488.151} C_VEL
LIN {X 0,Y 432.302,Z 117.259,A -85,B 0,C 180,E1 -9491.801,E2 -9491.801} C_VEL
LIN {X 0,Y 432.332,Z 117.254,A -85,B 0,C 180,E1 -9494.348,E2 -9494.348} C_VEL
LIN {X 0,Y 432.301,Z 117.258,A -85,B 0,C 180,E1 -9497.019,E2 -9497.019} C_VEL
LIN {X 0,Y 432.289,Z 117.262,A -85,B 0,C 180,E1 -9499.828,E2 -9499.828} C_VEL
LIN {X 0,Y 432.304,Z 117.262,A -85,B 0,C 180,E1 -9503.022,E2 -9503.022} C_VEL
LIN {X 0,Y 432.332,Z 117.257,A -85,B 0,C 180,E1 -9506.002,E2 -9506.002} C_VEL
LIN {X 0,Y 432.346,Z 117.256,A -85,B 0,C 180,E1 -9509.49,E2 -9509.49} C_VEL
LIN {X 0,Y 432.365,Z 117.356,A -85,B 0,C 180,E1 -9511.182,E2 -9511.182} C_VEL
LIN {X 0,Y 434.302,Z 122.543,A -85,B 0,C 180,E1 -9512.219,E2 -9512.219} C_VEL
LIN {X 0,Y 439.748,Z 132.102,A -85,B 0,C 180,E1 -9513.124,E2 -9513.124} C_VEL
LIN {X 0,Y 444.544,Z 141.754,A -85,B 0,C 180,E1 -9513.891,E2 -9513.891} C_VEL
LIN {X 0,Y 446.545,Z 146.84,A -85,B 0,C 180,E1 -9514.222,E2 -9514.222} C_VEL
LIN {X 0,Y 442.794,Z 231.106,A -85,B 0,C 180,E1 -9516.188,E2 -9516.188} C_VEL
LIN {X 0,Y 440.947,Z 287.508,A -85,B 0,C 180,E1 -9517.448,E2 -9517.448} C_VEL
LIN {X 0,Y 440.316,Z 303.645,A -85,B 0,C 180,E1 -9517.996,E2 -9517.996} C_VEL
LIN {X 0,Y 439.563,Z 318.089,A -85,B 0,C 180,E1 -9518.67,E2 -9518.67} C_VEL
LIN {X 0,Y 438.752,Z 331.776,A -85,B 0,C 180,E1 -9519.489,E2 -9519.489} C_VEL
LIN {X 0,Y 437.74,Z 346.017,A -85,B 0,C 180,E1 -9520.54,E2 -9520.54} C_VEL
LIN {X 0,Y 436.675,Z 359.09,A -85,B 0,C 180,E1 -9521.726,E2 -9521.726} C_VEL
LIN {X 0,Y 435.726,Z 369.808,A -85,B 0,C 180,E1 -9522.881,E2 -9522.881} C_VEL
LIN {X 0,Y 434.884,Z 380.782,A -85,B 0,C 180,E1 -9524.295,E2 -9524.295} C_VEL
LIN {X 0,Y 433.956,Z 391.467,A -85,B 0,C 180,E1 -9525.941,E2 -9525.941} C_VEL
LIN {X 0,Y 433.163,Z 400.292,A -85,B 0,C 180,E1 -9527.586,E2 -9527.586} C_VEL
LIN {X 0,Y 432.621,Z 407.603,A -85,B 0,C 180,E1 -9529.233,E2 -9529.233} C_VEL
LIN {X 0,Y 432.133,Z 414.337,A -85,B 0,C 180,E1 -9531.112,E2 -9531.112} C_VEL
LIN {X 0,Y 431.849,Z 418.349,A -85,B 0,C 180,E1 -9532.519,E2 -9532.519} C_VEL
LIN {X 0,Y 431.541,Z 422.525,A -85,B 0,C 180,E1 -9534.393,E2 -9534.393} C_VEL
LIN {X 0,Y 431.505,Z 425.382,A -85,B 0,C 180,E1 -9536.265,E2 -9536.265} C_VEL
LIN {X 0,Y 431.366,Z 427.015,A -85,B 0,C 180,E1 -9538.133,E2 -9538.133} C_VEL
LIN {X 0,Y 431.287,Z 427.437,A -85,B 0,C 180,E1 -9540,E2 -9540} C_VEL
LIN {X 0,Y 431.309,Z 426.638,A -85,B 0,C 180,E1 -9541.868,E2 -9541.868} C_VEL
LIN {X 0,Y 431.443,Z 424.594,A -85,B 0,C 180,E1 -9543.736,E2 -9543.736} C_VEL
LIN {X 0,Y 431.529,Z 421.294,A -85,B 0,C 180,E1 -9545.608,E2 -9545.608} C_VEL
LIN {X 0,Y 431.694,Z 416.667,A -85,B 0,C 180,E1 -9547.484,E2 -9547.484} C_VEL
LIN {X 0,Y 431.972,Z 410.601,A -85,B 0,C 180,E1 -9549.364,E2 -9549.364} C_VEL
LIN {X 0,Y 432.449,Z 402.92,A -85,B 0,C 180,E1 -9551.246,E2 -9551.246} C_VEL
LIN {X 0,Y 432.876,Z 394.684,A -85,B 0,C 180,E1 -9552.891,E2 -9552.891} C_VEL
LIN {X 0,Y 433.622,Z 384.674,A -85,B 0,C 180,E1 -9554.55,E2 -9554.55} C_VEL
LIN {X 0,Y 434.372,Z 374.434,A -85,B 0,C 180,E1 -9555.966,E2 -9555.966} C_VEL
LIN {X 0,Y 435.232,Z 362.847,A -85,B 0,C 180,E1 -9557.315,E2 -9557.315} C_VEL
LIN {X 0,Y 436.081,Z 350.055,A -85,B 0,C 180,E1 -9558.56,E2 -9558.56} C_VEL
LIN {X 0,Y 436.935,Z 336.868,A -85,B 0,C 180,E1 -9559.62,E2 -9559.62} C_VEL
LIN {X 0,Y 437.761,Z 322.447,A -85,B 0,C 180,E1 -9560.561,E2 -9560.561} C_VEL
LIN {X 0,Y 438.488,Z 307.519,A -85,B 0,C 180,E1 -9561.324,E2 -9561.324} C_VEL
LIN {X 0,Y 439.062,Z 292.192,A -85,B 0,C 180,E1 -9561.911,E2 -9561.911} C_VEL
LIN {X 0,Y 439.472,Z 276.527,A -85,B 0,C 180,E1 -9562.322,E2 -9562.322} C_VEL
LIN {X 0,Y 442.369,Z 148.375,A -85,B 0,C 180,E1 -9564.815,E2 -9564.815} C_VEL
LIN {X 0,Y 442.473,Z 142.942,A -85,B 0,C 180,E1 -9564.925,E2 -9564.925} C_VEL
LIN {X 0,Y 433.933,Z 121.414,A -85,B 0,C 180,E1 -9565.84,E2 -9565.84} C_VEL
LIN {X 0,Y 432.377,Z 117.253,A -85,B 0,C 180,E1 -9566.032,E2 -9566.032} C_VEL
LIN {X 0,Y 432.329,Z 117.257,A -85,B 0,C 180,E1 -9569.189,E2 -9569.189} C_VEL
LIN {X 0,Y 432.323,Z 117.256,A -85,B 0,C 180,E1 -9572.443,E2 -9572.443} C_VEL
LIN {X 0,Y 432.338,Z 117.257,A -85,B 0,C 180,E1 -9575.818,E2 -9575.818} C_VEL
LIN {X 0,Y 432.304,Z 117.263,A -85,B 0,C 180,E1 -9579.348,E2 -9579.348} C_VEL
LIN {X 0,Y 432.307,Z 117.26,A -85,B 0,C 180,E1 -9581.801,E2 -9581.801} C_VEL
LIN {X 0,Y 432.335,Z 117.249,A -85,B 0,C 180,E1 -9584.348,E2 -9584.348} C_VEL
LIN {X 0,Y 432.304,Z 117.241,A -85,B 0,C 180,E1 -9587.019,E2 -9587.019} C_VEL
LIN {X 0,Y 432.31,Z 117.258,A -85,B 0,C 180,E1 -9589.825,E2 -9589.825} C_VEL
LIN {X 0,Y 432.307,Z 117.252,A -85,B 0,C 180,E1 -9593.022,E2 -9593.022} C_VEL
LIN {X 0,Y 432.335,Z 117.25,A -85,B 0,C 180,E1 -9596.002,E2 -9596.002} C_VEL
LIN {X 0,Y 432.343,Z 117.247,A -85,B 0,C 180,E1 -9599.492,E2 -9599.492} C_VEL
LIN {X 0,Y 432.337,Z 117.25,A -85,B 0,C 180,E1 -9601.873,E2 -9601.873} C_VEL
LIN {X 0,Y 432.325,Z 117.251,A -85,B 0,C 180,E1 -9604.997,E2 -9604.997} C_VEL
LIN {X 0,Y 432.358,Z 117.252,A -85,B 0,C 180,E1 -9608.046,E2 -9608.046} C_VEL
LIN {X 0,Y 432.384,Z 117.25,A -85,B 0,C 180,E1 -9611.029,E2 -9611.029} C_VEL
LIN {X 0,Y 432.371,Z 117.245,A -85,B 0,C 180,E1 -9613.695,E2 -9613.695} C_VEL
LIN {X 0,Y 431.759,Z 117.327,A -85,B 0,C 180,E1 -9614.472,E2 -9614.472} C_VEL
LIN {X 0,Y 428.974,Z 117.675,A -85,B 0,C 180,E1 -9615.736,E2 -9615.736} C_VEL
LIN {X 0,Y 426.567,Z 117.974,A -85,B 0,C 180,E1 -9616.755,E2 -9616.755} C_VEL
LIN {X 0,Y 425.496,Z 118.106,A -85,B 0,C 180,E1 -9617.542,E2 -9617.542} C_VEL
LIN {X 0,Y 425.391,Z 118.118,A -85,B 0,C 180,E1 -9617.809,E2 -9617.809} C_VEL
LIN {X 0,Y 425.399,Z 118.119,A -85,B 0,C 180,E1 -9621.449,E2 -9621.449} C_VEL
LIN {X 0,Y 425.508,Z 118.109,A -85,B 0,C 180,E1 -9624.313,E2 -9624.313} C_VEL
LIN {X 0,Y 425.366,Z 118.289,A -85,B 0,C 180,E1 -9626.566,E2 -9626.566} C_VEL
LIN {X 0,Y 427.865,Z 127.383,A -85,B 0,C 180,E1 -9628.117,E2 -9628.117} C_VEL
LIN {X 0,Y 431.006,Z 141.544,A -85,B 0,C 180,E1 -9630.467,E2 -9630.467} C_VEL
LIN {X 0,Y 431.166,Z 143.135,A -85,B 0,C 180,E1 -9630.686,E2 -9630.686} C_VEL
LIN {X 0,Y 436.874,Z 169.78,A -85,B 0,C 180,E1 -9631.526,E2 -9631.526} C_VEL
LIN {X 0,Y 434.475,Z 309.505,A -85,B 0,C 180,E1 -9633.913,E2 -9633.913} C_VEL
LIN {X 0,Y 433.928,Z 324.799,A -85,B 0,C 180,E1 -9634.354,E2 -9634.354} C_VEL
LIN {X 0,Y 433.218,Z 339.089,A -85,B 0,C 180,E1 -9634.944,E2 -9634.944} C_VEL
LIN {X 0,Y 432.336,Z 352.908,A -85,B 0,C 180,E1 -9635.693,E2 -9635.693} C_VEL
LIN {X 0,Y 431.302,Z 367.041,A -85,B 0,C 180,E1 -9636.667,E2 -9636.667} C_VEL
LIN {X 0,Y 430.203,Z 379.763,A -85,B 0,C 180,E1 -9637.746,E2 -9637.746} C_VEL
LIN {X 0,Y 429.06,Z 392.577,A -85,B 0,C 180,E1 -9639.071,E2 -9639.071} C_VEL
LIN {X 0,Y 428.044,Z 403.358,A -85,B 0,C 180,E1 -9640.405,E2 -9640.405} C_VEL
LIN {X 0,Y 427.069,Z 413.343,A -85,B 0,C 180,E1 -9641.871,E2 -9641.871} C_VEL
LIN {X 0,Y 426.27,Z 422.131,A -85,B 0,C 180,E1 -9643.406,E2 -9643.406} C_VEL
LIN {X 0,Y 425.521,Z 430.14,A -85,B 0,C 180,E1 -9645.078,E2 -9645.078} C_VEL
LIN {X 0,Y 425.012,Z 437.085,A -85,B 0,C 180,E1 -9646.84,E2 -9646.84} C_VEL
LIN {X 0,Y 424.577,Z 443.327,A -85,B 0,C 180,E1 -9648.817,E2 -9648.817} C_VEL
LIN {X 0,Y 424.29,Z 448.229,A -85,B 0,C 180,E1 -9650.863,E2 -9650.863} C_VEL
LIN {X 0,Y 424.085,Z 450.923,A -85,B 0,C 180,E1 -9652.406,E2 -9652.406} C_VEL
LIN {X 0,Y 423.957,Z 453.341,A -85,B 0,C 180,E1 -9654.483,E2 -9654.483} C_VEL
LIN {X 0,Y 423.907,Z 454.384,A -85,B 0,C 180,E1 -9656.592,E2 -9656.592} C_VEL
LIN {X 0,Y 423.951,Z 454.008,A -85,B 0,C 180,E1 -9658.734,E2 -9658.734} C_VEL
LIN {X 0,Y 424.065,Z 452.138,A -85,B 0,C 180,E1 -9660.915,E2 -9660.915} C_VEL
LIN {X 0,Y 424.17,Z 450.124,A -85,B 0,C 180,E1 -9662.326,E2 -9662.326} C_VEL
LIN {X 0,Y 424.446,Z 446.252,A -85,B 0,C 180,E1 -9664.262,E2 -9664.262} C_VEL
LIN {X 0,Y 424.743,Z 441.188,A -85,B 0,C 180,E1 -9666.144,E2 -9666.144} C_VEL
LIN {X 0,Y 425.222,Z 434.824,A -85,B 0,C 180,E1 -9668,E2 -9668} C_VEL
LIN {X 0,Y 425.894,Z 427.238,A -85,B 0,C 180,E1 -9669.79,E2 -9669.79} C_VEL
LIN {X 0,Y 426.746,Z 418.335,A -85,B 0,C 180,E1 -9671.519,E2 -9671.519} C_VEL
LIN {X 0,Y 427.773,Z 408.213,A -85,B 0,C 180,E1 -9673.147,E2 -9673.147} C_VEL
LIN {X 0,Y 428.852,Z 396.988,A -85,B 0,C 180,E1 -9674.649,E2 -9674.649} C_VEL
LIN {X 0,Y 429.999,Z 384.981,A -85,B 0,C 180,E1 -9675.984,E2 -9675.984} C_VEL
LIN {X 0,Y 431.223,Z 371.985,A -85,B 0,C 180,E1 -9677.172,E2 -9677.172} C_VEL
LIN {X 0,Y 432.316,Z 358.211,A -85,B 0,C 180,E1 -9678.2,E2 -9678.2} C_VEL
LIN {X 0,Y 433.308,Z 343.967,A -85,B 0,C 180,E1 -9679.044,E2 -9679.044} C_VEL
LIN {X 0,Y 434.167,Z 329.135,A -85,B 0,C 180,E1 -9679.714,E2 -9679.714} C_VEL
LIN {X 0,Y 434.776,Z 314.791,A -85,B 0,C 180,E1 -9680.181,E2 -9680.181} C_VEL
LIN {X 0,Y 435.129,Z 297.821,A -85,B 0,C 180,E1 -9680.533,E2 -9680.533} C_VEL
LIN {X 0,Y 437.398,Z 164.513,A -85,B 0,C 180,E1 -9682.815,E2 -9682.815} C_VEL
LIN {X 0,Y 434.052,Z 146.456,A -85,B 0,C 180,E1 -9683.376,E2 -9683.376} C_VEL
LIN {X 0,Y 432.098,Z 141.604,A -85,B 0,C 180,E1 -9683.618,E2 -9683.618} C_VEL
LIN {X 0,Y 427.852,Z 126.275,A -85,B 0,C 180,E1 -9685.743,E2 -9685.743} C_VEL
LIN {X 0,Y 425.302,Z 118.132,A -85,B 0,C 180,E1 -9686.918,E2 -9686.918} C_VEL
LIN {X 0,Y 425.293,Z 118.13,A -85,B 0,C 180,E1 -9690.28,E2 -9690.28} C_VEL
LIN {X 0,Y 425.369,Z 118.166,A -85,B 0,C 180,E1 -9693.66,E2 -9693.66} C_VEL
LIN {X 0,Y 427.229,Z 123.021,A -85,B 0,C 180,E1 -9693.875,E2 -9693.875} C_VEL
LIN {X 0,Y 434.674,Z 140.827,A -85,B 0,C 180,E1 -9694.678,E2 -9694.678} C_VEL
LIN {X 0,Y 436.053,Z 144.815,A -85,B 0,C 180,E1 -9694.838,E2 -9694.838} C_VEL
LIN {X 0,Y 432.598,Z 283.895,A -85,B 0,C 180,E1 -9697.637,E2 -9697.637} C_VEL
LIN {X 0,Y 432.093,Z 299.426,A -85,B 0,C 180,E1 -9698.135,E2 -9698.135} C_VEL
LIN {X 0,Y 431.42,Z 314.564,A -85,B 0,C 180,E1 -9698.811,E2 -9698.811} C_VEL
LIN {X 0,Y 430.666,Z 328.079,A -85,B 0,C 180,E1 -9699.585,E2 -9699.585} C_VEL
LIN {X 0,Y 429.834,Z 341.522,A -85,B 0,C 180,E1 -9700.54,E2 -9700.54} C_VEL
LIN {X 0,Y 428.917,Z 355.264,A -85,B 0,C 180,E1 -9701.737,E2 -9701.737} C_VEL
LIN {X 0,Y 427.986,Z 367.748,A -85,B 0,C 180,E1 -9703.053,E2 -9703.053} C_VEL
LIN {X 0,Y 427.15,Z 379.134,A -85,B 0,C 180,E1 -9704.492,E2 -9704.492} C_VEL
LIN {X 0,Y 426.42,Z 388.744,A -85,B 0,C 180,E1 -9705.93,E2 -9705.93} C_VEL
LIN {X 0,Y 425.799,Z 398.13,A -85,B 0,C 180,E1 -9707.609,E2 -9707.609} C_VEL
LIN {X 0,Y 425.217,Z 405.893,A -85,B 0,C 180,E1 -9709.284,E2 -9709.284} C_VEL
LIN {X 0,Y 424.875,Z 412.281,A -85,B 0,C 180,E1 -9710.959,E2 -9710.959} C_VEL
LIN {X 0,Y 424.553,Z 418.119,A -85,B 0,C 180,E1 -9712.868,E2 -9712.868} C_VEL
LIN {X 0,Y 424.489,Z 421.569,A -85,B 0,C 180,E1 -9714.299,E2 -9714.299} C_VEL
LIN {X 0,Y 424.388,Z 424.984,A -85,B 0,C 180,E1 -9716.202,E2 -9716.202} C_VEL
LIN {X 0,Y 424.246,Z 427.119,A -85,B 0,C 180,E1 -9718.101,E2 -9718.101} C_VEL
LIN {X 0,Y 424.213,Z 428.026,A -85,B 0,C 180,E1 -9720,E2 -9720} C_VEL
LIN {X 0,Y 424.313,Z 427.718,A -85,B 0,C 180,E1 -9721.898,E2 -9721.898} C_VEL
LIN {X 0,Y 424.46,Z 426.198,A -85,B 0,C 180,E1 -9723.797,E2 -9723.797} C_VEL
LIN {X 0,Y 424.509,Z 423.453,A -85,B 0,C 180,E1 -9725.701,E2 -9725.701} C_VEL
LIN {X 0,Y 424.812,Z 419.396,A -85,B 0,C 180,E1 -9727.605,E2 -9727.605} C_VEL
LIN {X 0,Y 425.287,Z 413.93,A -85,B 0,C 180,E1 -9729.512,E2 -9729.512} C_VEL
LIN {X 0,Y 425.806,Z 406.935,A -85,B 0,C 180,E1 -9731.423,E2 -9731.423} C_VEL
LIN {X 0,Y 426.44,Z 399.374,A -85,B 0,C 180,E1 -9733.097,E2 -9733.097} C_VEL
LIN {X 0,Y 427.384,Z 390.222,A -85,B 0,C 180,E1 -9734.767,E2 -9734.767} C_VEL
LIN {X 0,Y 428.213,Z 380.89,A -85,B 0,C 180,E1 -9736.201,E2 -9736.201} C_VEL
LIN {X 0,Y 429.245,Z 369.81,A -85,B 0,C 180,E1 -9737.632,E2 -9737.632} C_VEL
LIN {X 0,Y 430.343,Z 357.654,A -85,B 0,C 180,E1 -9738.94,E2 -9738.94} C_VEL
LIN {X 0,Y 431.407,Z 344.382,A -85,B 0,C 180,E1 -9740.129,E2 -9740.129} C_VEL
LIN {X 0,Y 432.455,Z 331.453,A -85,B 0,C 180,E1 -9741.073,E2 -9741.073} C_VEL
LIN {X 0,Y 433.339,Z 317.57,A -85,B 0,C 180,E1 -9741.902,E2 -9741.902} C_VEL
LIN {X 0,Y 434.177,Z 302.693,A -85,B 0,C 180,E1 -9742.59,E2 -9742.59} C_VEL
LIN {X 0,Y 434.771,Z 287.535,A -85,B 0,C 180,E1 -9743.11,E2 -9743.11} C_VEL
LIN {X 0,Y 437.742,Z 210.987,A -85,B 0,C 180,E1 -9744.894,E2 -9744.894} C_VEL
LIN {X 0,Y 440.776,Z 150.035,A -85,B 0,C 180,E1 -9746.398,E2 -9746.398} C_VEL
LIN {X 0,Y 435.495,Z 139.543,A -85,B 0,C 180,E1 -9747.271,E2 -9747.271} C_VEL
LIN {X 0,Y 429.921,Z 130.028,A -85,B 0,C 180,E1 -9748.237,E2 -9748.237} C_VEL
LIN {X 0,Y 428.018,Z 126.821,A -85,B 0,C 180,E1 -9748.603,E2 -9748.603} C_VEL
LIN {X 0,Y 425.949,Z 120.403,A -85,B 0,C 180,E1 -9750.909,E2 -9750.909} C_VEL
LIN {X 0,Y 425.278,Z 118.139,A -85,B 0,C 180,E1 -9751.856,E2 -9751.856} C_VEL
LIN {X 0,Y 425.294,Z 118.136,A -85,B 0,C 180,E1 -9755.336,E2 -9755.336} C_VEL
LIN {X 0,Y 425.28,Z 118.138,A -85,B 0,C 180,E1 -9758.9,E2 -9758.9} C_VEL
LIN {X 0,Y 425.255,Z 118.139,A -85,B 0,C 180,E1 -9762.655,E2 -9762.655} C_VEL
LIN {X 0,Y 425.284,Z 118.136,A -85,B 0,C 180,E1 -9765.283,E2 -9765.283} C_VEL
LIN {X 0,Y 425.246,Z 118.142,A -85,B 0,C 180,E1 -9768.618,E2 -9768.618} C_VEL
LIN {X 0,Y 425.279,Z 118.138,A -85,B 0,C 180,E1 -9771.099,E2 -9771.099} C_VEL
LIN {X 0,Y 425.285,Z 118.224,A -85,B 0,C 180,E1 -9772.531,E2 -9772.531} C_VEL
LIN {X 0,Y 427.19,Z 123.742,A -85,B 0,C 180,E1 -9774.401,E2 -9774.401} C_VEL
LIN {X 0,Y 429.6,Z 131.184,A -85,B 0,C 180,E1 -9776.546,E2 -9776.546} C_VEL
LIN {X 0,Y 432.116,Z 140.824,A -85,B 0,C 180,E1 -9778.894,E2 -9778.894} C_VEL
LIN {X 0,Y 433.515,Z 147.689,A -85,B 0,C 180,E1 -9780.366,E2 -9780.366} C_VEL
LIN {X 0,Y 432.482,Z 156.881,A -85,B 0,C 180,E1 -9781.93,E2 -9781.93} C_VEL
LIN {X 0,Y 436.172,Z 174.478,A -85,B 0,C 180,E1 -9782.874,E2 -9782.874} C_VEL
LIN {X 0,Y 438.41,Z 188.626,A -85,B 0,C 180,E1 -9783.516,E2 -9783.516} C_VEL
LIN {X 0,Y 439.308,Z 197.744,A -85,B 0,C 180,E1 -9783.862,E2 -9783.862} C_VEL
LIN {X 0,Y 435.656,Z 281.133,A -85,B 0,C 180,E1 -9785.836,E2 -9785.836} C_VEL
LIN {X 0,Y 433.995,Z 329.283,A -85,B 0,C 180,E1 -9786.941,E2 -9786.941} C_VEL
LIN {X 0,Y 432.92,Z 346.165,A -85,B 0,C 180,E1 -9787.52,E2 -9787.52} C_VEL
LIN {X 0,Y 431.805,Z 365.684,A -85,B 0,C 180,E1 -9788.375,E2 -9788.375} C_VEL
LIN {X 0,Y 430.804,Z 380.24,A -85,B 0,C 180,E1 -9789.217,E2 -9789.217} C_VEL
LIN {X 0,Y 429.873,Z 393.264,A -85,B 0,C 180,E1 -9790.169,E2 -9790.169} C_VEL
LIN {X 0,Y 428.817,Z 405.354,A -85,B 0,C 180,E1 -9791.238,E2 -9791.238} C_VEL
LIN {X 0,Y 427.861,Z 416.785,A -85,B 0,C 180,E1 -9792.457,E2 -9792.457} C_VEL
LIN {X 0,Y 426.771,Z 428.744,A -85,B 0,C 180,E1 -9793.988,E2 -9793.988} C_VEL
LIN {X 0,Y 426.023,Z 438.129,A -85,B 0,C 180,E1 -9795.429,E2 -9795.429} C_VEL
LIN {X 0,Y 425.261,Z 447.649,A -85,B 0,C 180,E1 -9797.175,E2 -9797.175} C_VEL
LIN {X 0,Y 424.809,Z 455.914,A -85,B 0,C 180,E1 -9799.032,E2 -9799.032} C_VEL
LIN {X 0,Y 424.396,Z 462.775,A -85,B 0,C 180,E1 -9800.949,E2 -9800.949} C_VEL
LIN {X 0,Y 424.279,Z 468.133,A -85,B 0,C 180,E1 -9802.863,E2 -9802.863} C_VEL
LIN {X 0,Y 424.171,Z 471.2,A -85,B 0,C 180,E1 -9804.295,E2 -9804.295} C_VEL
LIN {X 0,Y 424.102,Z 474.215,A -85,B 0,C 180,E1 -9806.199,E2 -9806.199} C_VEL
LIN {X 0,Y 424.183,Z 476.013,A -85,B 0,C 180,E1 -9808.101,E2 -9808.101} C_VEL
LIN {X 0,Y 424.088,Z 476.617,A -85,B 0,C 180,E1 -9810,E2 -9810} C_VEL
LIN {X 0,Y 424.182,Z 476.005,A -85,B 0,C 180,E1 -9811.899,E2 -9811.899} C_VEL
LIN {X 0,Y 424.109,Z 474.184,A -85,B 0,C 180,E1 -9813.801,E2 -9813.801} C_VEL
LIN {X 0,Y 424.184,Z 471.134,A -85,B 0,C 180,E1 -9815.705,E2 -9815.705} C_VEL
LIN {X 0,Y 424.297,Z 466.78,A -85,B 0,C 180,E1 -9817.615,E2 -9817.615} C_VEL
LIN {X 0,Y 424.451,Z 461.013,A -85,B 0,C 180,E1 -9819.531,E2 -9819.531} C_VEL
LIN {X 0,Y 424.891,Z 453.675,A -85,B 0,C 180,E1 -9821.449,E2 -9821.449} C_VEL
LIN {X 0,Y 425.355,Z 445.542,A -85,B 0,C 180,E1 -9823.174,E2 -9823.174} C_VEL
LIN {X 0,Y 426.06,Z 436.199,A -85,B 0,C 180,E1 -9824.814,E2 -9824.814} C_VEL
LIN {X 0,Y 426.884,Z 426.404,A -85,B 0,C 180,E1 -9826.253,E2 -9826.253} C_VEL
LIN {X 0,Y 427.797,Z 414.94,A -85,B 0,C 180,E1 -9827.666,E2 -9827.666} C_VEL
LIN {X 0,Y 428.747,Z 403.024,A -85,B 0,C 180,E1 -9828.889,E2 -9828.889} C_VEL
LIN {X 0,Y 429.811,Z 390.392,A -85,B 0,C 180,E1 -9829.958,E2 -9829.958} C_VEL
LIN {X 0,Y 430.791,Z 376.552,A -85,B 0,C 180,E1 -9830.908,E2 -9830.908} C_VEL
LIN {X 0,Y 431.721,Z 361.874,A -85,B 0,C 180,E1 -9831.692,E2 -9831.692} C_VEL
LIN {X 0,Y 432.402,Z 346.792,A -85,B 0,C 180,E1 -9832.291,E2 -9832.291} C_VEL
